                       // ================================================
                       // Proceed the reactive power for each phase
                       // ================================================
                       #Driver_Data.Q_L1_max := #V_DP_Meas_Min_Max.Q_L1_Max;
                       #Driver_Data.Q_L1_min := #V_DP_Meas_Min_Max.Q_L1_Min;
                       #Driver_Data.Q_L2_max := #V_DP_Meas_Min_Max.Q_L2_Max;
                       #Driver_Data.Q_L2_min := #V_DP_Meas_Min_Max.Q_L2_Min;
                       #Driver_Data.Q_L3_max := #V_DP_Meas_Min_Max.Q_L3_Max;
                       #Driver_Data.Q_L3_min := #V_DP_Meas_Min_Max.Q_L3_Min;
                       #Driver_Data.Q_Total_max := #V_DP_Meas_Min_Max.Q_Total_Max;
                       #Driver_Data.Q_Total_min := #V_DP_Meas_Min_Max.Q_Total_Min;

                       // ================================================
                       // Proceed the effective power for each phase
                       // ================================================
                       #Driver_Data.P_L1_max := #V_DP_Meas_Min_Max.P_L1_Max;
                       #Driver_Data.P_L1_min := #V_DP_Meas_Min_Max.P_L1_Min;
                       #Driver_Data.P_L2_max := #V_DP_Meas_Min_Max.P_L2_Max;
                       #Driver_Data.P_L2_min := #V_DP_Meas_Min_Max.P_L2_Min;
                       #Driver_Data.P_L3_max := #V_DP_Meas_Min_Max.P_L3_Max;
                       #Driver_Data.P_L3_min := #V_DP_Meas_Min_Max.P_L3_Min;
                       #Driver_Data.P_Total_max := #V_DP_Meas_Min_Max.P_Total_Max;
                       #Driver_Data.P_Total_min := #V_DP_Meas_Min_Max.P_Total_Min;

                       // Go back to the main state and wait for a new request
                       #Sm_State_Next := #SM_IDLE;
                   ELSE
                       ; // Reading still in progress
                   END_IF;
           END_CASE;

           // Set information for the visualization block
           #Driver_Data.Read_Value := #Automatic_Update;
           #Driver_Data.Driver_Error := BOOL_TO_INT(#Error_Code <> 0);
           #Driver_Data.Connection_Type := #Connection_Type;

           // Store the value for edge detection
           #Start_Acyclic_HMI_Old := #HMI_Bits_Internal.Start_Acyclic;
           #Reset_Energy_Old := #Reset_Energy_Counter;
           #Reset_Energy_HMI_Old := #HMI_Bits_Internal.Reset_Energy_Meter;
           #Reset_Min_Max_Old := #Reset_Min_Max;
           #Reset_Min_Max_HMI_Old := #HMI_Bits_Internal.Reset_min_max_Data;

       END_IF;
END_FUNCTION_BLOCK

FUNCTION_BLOCK "LProcPAC-Conversion"   // FB1743, SCL
TITLE = LProcPAC-Conversion
{ S7_Optimized_Access := 'TRUE' }
AUTHOR : CSTAAL
VERSION : 2.0
// stored: AutoNumber false, IsIECCheckEnabled false, IsRetainMemResEnabled false, MemoryReserve 100, SetENOAutomatically False, UDAEnableTagReadback false
   VAR_INPUT
      id_hdword { ExternalAccessible := 'False'; ExternalVisible := 'False'; ExternalWritable := 'False'} : DWord := DWORD#16#0000_0000;   // highdword of the 64Bit number
      id_ldword { ExternalAccessible := 'False'; ExternalVisible := 'False'; ExternalWritable := 'False'} : DWord := DWORD#16#0000_0000;   // lowdword of the 64Bit number
   END_VAR
   VAR_OUTPUT
      FINE { ExternalAccessible := 'False'; ExternalVisible := 'False'; ExternalWritable := 'False'} : DInt := 0;   // counter value fine
      RAW { ExternalAccessible := 'False'; ExternalVisible := 'False'; ExternalWritable := 'False'} : DInt := 0;   // counter value raw
      ERROR { ExternalAccessible := 'False'; ExternalVisible := 'False'; ExternalWritable := 'False'} : Word := WORD#16#0000;   // error word of the function block
   END_VAR
   VAR DB_SPECIFIC
      sCounterval { ExternalAccessible := 'False'; ExternalVisible := 'False'; ExternalWritable := 'False'} : Struct   // 64Bit structure
         hdword { ExternalAccessible := 'False'; ExternalVisible := 'False'; ExternalWritable := 'False'} : DWord := DWORD#16#0000_0000;   // highdword of the 64Bit number
         ldword { ExternalAccessible := 'False'; ExternalVisible := 'False'; ExternalWritable := 'False'} : DWord := DWORD#16#0000_0000;   // lowdword of the 64Bit number
      END_STRUCT;
   END_VAR
   VAR
      vwords AT sCounterval : Struct   // AT sCounterval : STRUCT
         HDHW : Word;   // highword of the highdword of the 64Bit number
         HDLW : Word;   // lowword of the highdword of the 64Bit number
         LDHW : Word;   // highword of the lowdword of the 64Bit number
         LDLW : Word;   // lowword of the lowdword of the 64Bit number
      END_STRUCT;
      sVZ { ExternalAccessible := 'False'; ExternalVisible := 'False'; ExternalWritable := 'False'} : Word := WORD#16#0000;   // algebraic sign of the 64Bit number
      sCH { ExternalAccessible := 'False'; ExternalVisible := 'False'; ExternalWritable := 'False'} : Word := WORD#16#0000;   // exponent of the 64Bit number
      sExp { ExternalAccessible := 'False'; ExternalVisible := 'False'; ExternalWritable := 'False'} : Int := 0;   // exponent of the 64Bit number
      sResDiv { ExternalAccessible := 'False'; ExternalVisible := 'False'; ExternalWritable := 'False'} : DWord := DWORD#16#0000_0000;   // result of division
      sDivision { ExternalAccessible := 'False'; ExternalVisible := 'False'; ExternalWritable := 'False'} : DWord := DWORD#16#0000_0000;   // dword for division of 1.000.000.000
      sFINE { ExternalAccessible := 'False'; ExternalVisible := 'False'; ExternalWritable := 'False'} : DInt := 0;   // static counter falue fine
      sRAW { ExternalAccessible := 'False'; ExternalVisible := 'False'; ExternalWritable := 'False'} : DInt := 0;   // static counter value raw
      sERROR { ExternalAccessible := 'False'; ExternalVisible := 'False'; ExternalWritable := 'False'} : Word := WORD#16#0000;   // static error word
      i { ExternalAccessible := 'False'; ExternalVisible := 'False'; ExternalWritable := 'False'} : Int := 0;   // loop counter
   END_VAR
   VAR CONSTANT
      cBIAS : Word := WORD#16#03FF;   // 03FFh --> 1023dez ... bias of the 64Bit number
      cVZmask : Word := WORD#16#8000;   // mask to seperate the algebraic sign
      cCHmask : Word := WORD#16#7FF0;   // mask to seperate the exponent field
      cMTmask : DWord := DWORD#16#000F_FFFF;   // mask to seperate the mantissa
      cMask : DWord := DWORD#16#0000_0001;   // general mask
      cNrGIGA : DInt := 1_000_000_000;   // 1.000.000.000(dez)
      cNrKILO : Int := 1000;   // 1.000(dez)
   END_VAR
BEGIN



   (***********************************************************************************************
   ********************************************  CODE  *******************************************
   ***********************************************************************************************)

   // initialization of internal variables
   // allocation of the two dwords of the energy counter value
   #sCounterval.hdword := #id_hdword;
   #sCounterval.ldword := #id_ldword;
   #sResDiv := dw#16#000000000;

   // seperate VZ (sign bit)
   #sVZ := #vwords.HDHW AND #cVZmask;

   // seperate CH (exponent field with offset(cBias))
   // seperate exponent of the 64Bit value
   #sCH := SHR(IN := (#vwords.HDHW AND #cCHmask), N := 4);
   #sExp := WORD_TO_INT(#sCH) - WORD_TO_INT(#cBIAS);

   // check the algebraic sign
   // negative counter values indicate an error
   IF #sVZ = #cVZmask
   THEN
       #sERROR := w#16#0001;
   ELSE
       // check the special case of the 0 value and the value < 1
       // the output values have the format dint --> 0,1 is not possible
       IF #sCH = w#16#0000 OR WORD_TO_INT(#sCH) < WORD_TO_INT(#cBIAS)
       THEN
           #sFINE := 0;
           #sRAW := 0;
       ELSE
           // **************************
           // ********** FINE **********
           // **************************

           // *** If the exponent is smaller than 29 the number is smaller than 1.000.000.000
           // *** You have to seperate the valid bits (sExp)of the mantissa
           // *** At the end you have to add the hidden 1 Bit
           IF #sExp < 29
           THEN
               IF #sExp < 20
               THEN
                   #sFINE := DWORD_TO_DINT(SHR(IN := (#sCounterval.hdword AND #cMTmask), N := 20 - #sExp) OR SHL(IN := #cMask, N := #sExp));

               ELSIF #sExp = 20
               THEN
                   #sFINE := DWORD_TO_DINT(#sCounterval.hdword AND #cMTmask OR SHL(IN := #cMask, N := 20));
               ELSE
                   #sFINE := DWORD_TO_DINT((SHL(IN := (#sCounterval.hdword AND #cMTmask), N := #sExp - 20) OR SHR(IN := #sCounterval.ldword, N := 32 - (#sExp - 20))) OR SHL(IN := #cMask, N := #sExp));
               END_IF;

               // *** If the exponent is 29 the number is between 536.870.912 and 1.073.741.823
               // *** You have to subtract 1.000.000.000 if it's bigger than 1.000.000.000
               // *** The result ist the fine counter value
           ELSIF #sExp = 29
           THEN
               IF DWORD_TO_DINT((SHL(IN := (#sCounterval.hdword AND #cMTmask), N := #sExp - 20) OR SHR(IN := #sCounterval.ldword, N := 32 - (#sExp - 20))) OR SHL(IN := #cMask, N := #sExp)) > #cNrGIGA
               THEN
                   #sFINE := DWORD_TO_DINT((SHL(IN := (#sCounterval.hdword AND #cMTmask), N := #sExp - 20) OR SHR(IN := #sCounterval.ldword, N := 32 - (#sExp - 20))) OR SHL(IN := #cMask, N := #sExp)) - #cNrGIGA;

               ELSIF DWORD_TO_DINT((SHL(IN := (#sCounterval.hdword AND #cMTmask), N := #sExp - 20) OR SHR(IN := #sCounterval.ldword, N := 32 - (#sExp - 20))) OR SHL(IN := #cMask, N := #sExp)) = #cNrGIGA
               THEN
                   #sFINE := 0;
               ELSE
                   #sFINE := DWORD_TO_DINT((SHL(IN := (#sCounterval.hdword AND #cMTmask), N := #sExp - 20) OR SHR(IN := #sCounterval.ldword, N := 32 - (#sExp - 20))) OR SHL(IN := #cMask, N := #sExp));
               END_IF;

               // *** If the exponent is bigger then 29 you have to divide the number by 1.000.000.000
               // *** the rest of the division is the fine counter value
           ELSE
               #sDivision := (SHL(IN := (#sCounterval.hdword AND #cMTmask), N := 9) OR SHR(IN := #sCounterval.ldword, N := 23)) OR SHL(IN := #cMask, N := 29);
               FOR #i := 0 TO #sExp - 29 DO
                   IF DWORD_TO_DINT(#sDivision) > #cNrGIGA OR DWORD_TO_DINT(#sDivision) = #cNrGIGA
                   THEN

                       #sDivision := DINT_TO_DWORD(DWORD_TO_DINT(#sDivision) - #cNrGIGA);
                       IF #i <> #sExp - 29
                       THEN
                           #sDivision := SHL(IN := #sDivision, N := 1) OR (SHR(IN := #sCounterval.ldword, N := 22 - #i) AND #cMask);
                       ELSE
                           ;
                       END_IF;

                       #sResDiv := SHL(IN := #sResDiv, N := 1) OR dw#16#00000001;
                   ELSE
                       IF #i <> #sExp - 29
                       THEN
                           #sDivision := SHL(IN := #sDivision, N := 1) OR (SHR(IN := #sCounterval.ldword, N := 22 - #i) AND #cMask);
                       ELSE
                           ;
                       END_IF;

                       #sResDiv := SHL(IN := #sResDiv, N := 1);
                   END_IF;

               END_FOR;

               #sFINE := DWORD_TO_DINT(#sDivision);

           END_IF;

           // **************************
           // ********** RAW ***********
           // **************************

           // Initialisation of sResDiv for new division
           #sResDiv := dw#16#00000000;

           // *** If the exponent is smaller than 9 the number is smaller than 1.000
           // *** The raw counter value is 0
           IF #sExp < 9
           THEN
               #sRAW := 0;

               // *** If the exponent is 9 the number is between 512 and 1.023
               // *** You have to subtract 1.000
               // *** The result ist the raw counter value
           ELSIF #sExp = 9
           THEN
               IF DWORD_TO_DINT(SHR(IN := (#sCounterval.hdword AND #cMTmask), N := 20 - #sExp) OR SHL(IN := #cMask, N := #sExp)) > #cNrKILO
               THEN
                   #sRAW := 1;
               ELSE
                   #sRAW := 0;
               END_IF;

               // *** If the exponent is bigger then 29 you have to divide the number by 1.000.000.000
               // *** the result of the division is the raw countervalue
           ELSE
               #sDivision := SHR(IN := (#sCounterval.hdword AND #cMTmask), N := 11) OR SHL(IN := #cMask, N := 9);
               FOR #i := 0 TO #sExp - 9 DO
                   IF DWORD_TO_DINT(#sDivision) > #cNrKILO OR DWORD_TO_DINT(#sDivision) = #cNrKILO
                   THEN

                       #sDivision := DINT_TO_DWORD(DWORD_TO_DINT(#sDivision) - #cNrKILO);
                       IF #i <> #sExp - 9
                       THEN
                           #sDivision := SHL(IN := #sDivision, N := 1);
                           IF #i <= 10
                           THEN
                               #sDivision := #sDivision OR (SHR(IN := #sCounterval.hdword, N := 11 - (#i + 1)) AND #cMask);
                           ELSE
                               #sDivision := #sDivision OR (SHR(IN := #sCounterval.ldword, N := 32 - ((#i + 1) - 11)) AND #cMask);
                           END_IF;

                       ELSE
                           ;
                       END_IF;

                       #sResDiv := SHL(IN := #sResDiv, N := 1) OR dw#16#00000001;
                   ELSE
                       IF #i <> #sExp - 9
                       THEN
                           #sDivision := SHL(IN := #sDivision, N := 1);
                           IF #i <= 10
                           THEN
                               #sDivision := #sDivision OR (SHR(IN := #sCounterval.hdword, N := 11 - (#i + 1)) AND #cMask);
                           ELSE
                               #sDivision := #sDivision OR (SHR(IN := #sCounterval.ldword, N := 32 - ((#i + 1) - 11)) AND #cMask);
                           END_IF;

                       ELSE
                           ;
                       END_IF;

                       #sResDiv := SHL(IN := #sResDiv, N := 1);
                   END_IF;

               END_FOR;

               #sRAW := DWORD_TO_DINT(#sResDiv);

           END_IF;

       END_IF;
       #sERROR := w#16#0000;
   END_IF;

   #FINE := #sFINE;
   #RAW := #sRAW;
   #ERROR := #sERROR;
END_FUNCTION_BLOCK

FUNCTION_BLOCK "LProcPAC-Visu"   // FB1742, SCL
TITLE = LProcPAC-Visu
{ S7_Optimized_Access := 'FALSE' }
AUTHOR : CSTAAL
VERSION : 2.0
// 20131213
// ======================================================================================================================
// ==========Short Description===========================================================================================
// ======================================================================================================================
// 
//   This function block is a interface between driver function block and WinCC. 
//   
// ======================================================================================================================
// ==========Dependencies(Abhängigkeit)==================================================================================
// ======================================================================================================================
// 
//   none
// 
// ======================================================================================================================
// ==========Change Log==================================================================================================
// ======================================================================================================================
// 
//       DATE    |   Version     |   NAME        |   CHANGE
//   ------------|---------------|---------------|--------------------------
//               |   v1.0        |   DirkTie     |   - First implementation 
//   ------------|---------------|---------------|--------------------------
//               |   v2.0        |   BaueChr     |   - bug fixes 
//   ------------|---------------|---------------|--------------------------
// 
// ======================================================================================================================
// ==========Know Issues=================================================================================================
// ======================================================================================================================
// 
//     - v2.0:
//             wrong connections of the energy counters to the outputs                 ... fixed 2014/08/22
//             extent the automatic change of the current unit over all phases            ... fixed 2014/08/22
//             extent driver_data structure (Connection_Type & Driver_error)            ... fixed 2014/08/22
//             change constant MAX_VALUE to 750 to define the correct scale end value    ... fixed 2014/08/25
//             new definition of the scale start value of reactive power if Qmin > 0    ... fixed 2014/08/25
// 
// ======================================================================================================================
// ==========Constant Definitions========================================================================================
// ======================================================================================================================
// stored: AutoNumber false, IsIECCheckEnabled false, SetENOAutomatically False, UDAEnableTagReadback false
   VAR_INPUT
      Add_Value_Count { ExternalAccessible := 'False'; ExternalVisible := 'False'; ExternalWritable := 'False'} : Int := 0;   // count of the user measurements
      AddValue_01 { ExternalAccessible := 'False'; ExternalVisible := 'False'; ExternalWritable := 'False'} : Real := 0.0;   // user measurements 01
      AddValue_02 { ExternalAccessible := 'False'; ExternalVisible := 'False'; ExternalWritable := 'False'} : Real := 0.0;   // user measurements 02
      AddValue_03 { ExternalAccessible := 'False'; ExternalVisible := 'False'; ExternalWritable := 'False'} : Real := 0.0;   // user measurements 03
      AddValue_04 { ExternalAccessible := 'False'; ExternalVisible := 'False'; ExternalWritable := 'False'} : Real := 0.0;   // user measurements 04
      AddValue_05 { ExternalAccessible := 'False'; ExternalVisible := 'False'; ExternalWritable := 'False'} : Real := 0.0;   // user measurements 05
      AddValue_06 { ExternalAccessible := 'False'; ExternalVisible := 'False'; ExternalWritable := 'False'} : Real := 0.0;   // user measurements 06
      AddValue_07 { ExternalAccessible := 'False'; ExternalVisible := 'False'; ExternalWritable := 'False'} : Real := 0.0;   // user measurements 07
      AddValue_08 { ExternalAccessible := 'False'; ExternalVisible := 'False'; ExternalWritable := 'False'} : Real := 0.0;   // user measurements 08
      AddValue_09 { ExternalAccessible := 'False'; ExternalVisible := 'False'; ExternalWritable := 'False'} : Real := 0.0;   // user measurements 09
      AddValue_10 { ExternalAccessible := 'False'; ExternalVisible := 'False'; ExternalWritable := 'False'} : Real := 0.0;   // user measurements 10
      AddValue_11 { ExternalAccessible := 'False'; ExternalVisible := 'False'; ExternalWritable := 'False'} : Real := 0.0;   // user measurements 11
      AddValue_12 { ExternalAccessible := 'False'; ExternalVisible := 'False'; ExternalWritable := 'False'} : Real := 0.0;   // user measurements 12
      Start_Acyclic { ExternalAccessible := 'False'; ExternalVisible := 'False'; ExternalWritable := 'False'} : Bool := FALSE;
      Start_Auto { ExternalAccessible := 'False'; ExternalVisible := 'False'; ExternalWritable := 'False'} : Bool := FALSE;
      Reset_min_max_Data { ExternalAccessible := 'False'; ExternalVisible := 'False'; ExternalWritable := 'False'} : Bool := FALSE;
      Reset_Energy_Meter { ExternalAccessible := 'False'; ExternalVisible := 'False'; ExternalWritable := 'False'} : Bool := FALSE;   // ================================================================================================================================inoutput variablen================================================================================================================================================================================================================
   END_VAR
   VAR_OUTPUT
      U_L1_L2 { ExternalAccessible := 'False'; ExternalVisible := 'False'; ExternalWritable := 'False'} : Real := 0.0;   // voltage L1-L2
      U_L2_L3 { ExternalAccessible := 'False'; ExternalVisible := 'False'; ExternalWritable := 'False'} : Real := 0.0;   // voltage L2-L3
      U_L3_L1 { ExternalAccessible := 'False'; ExternalVisible := 'False'; ExternalWritable := 'False'} : Real := 0.0;   // voltage L3-L1
      U_L1 { ExternalAccessible := 'False'; ExternalVisible := 'False'; ExternalWritable := 'False'} : Real := 0.0;   // voltage L1-N
      U_L2 { ExternalAccessible := 'False'; ExternalVisible := 'False'; ExternalWritable := 'False'} : Real := 0.0;   // voltage L2-N
      U_L3 { ExternalAccessible := 'False'; ExternalVisible := 'False'; ExternalWritable := 'False'} : Real := 0.0;   // voltage L3-N
      U_L1_L2_min { ExternalAccessible := 'False'; ExternalVisible := 'False'; ExternalWritable := 'False'} : Real := 0.0;   // minimum voltage U1
      U_L2_L3_min { ExternalAccessible := 'False'; ExternalVisible := 'False'; ExternalWritable := 'False'} : Real := 0.0;   // minimum voltage U2
      U_L3_L1_min { ExternalAccessible := 'False'; ExternalVisible := 'False'; ExternalWritable := 'False'} : Real := 0.0;
      U_L1_min { ExternalAccessible := 'False'; ExternalVisible := 'False'; ExternalWritable := 'False'} : Real := 0.0;   // minimum voltage U1
      U_L2_min { ExternalAccessible := 'False'; ExternalVisible := 'False'; ExternalWritable := 'False'} : Real := 0.0;   // minimum voltage U2
      U_L3_min { ExternalAccessible := 'False'; ExternalVisible := 'False'; ExternalWritable := 'False'} : Real := 0.0;   // minimum voltage U3
      U_L1_L2_max { ExternalAccessible := 'False'; ExternalVisible := 'False'; ExternalWritable := 'False'} : Real := 0.0;   // maximum voltage U1
      U_L2_L3_max { ExternalAccessible := 'False'; ExternalVisible := 'False'; ExternalWritable := 'False'} : Real := 0.0;   // maximum voltage U2
      U_L3_L1_max { ExternalAccessible := 'False'; ExternalVisible := 'False'; ExternalWritable := 'False'} : Real := 0.0;   // maximum voltage U3
      U_L1_max { ExternalAccessible := 'False'; ExternalVisible := 'False'; ExternalWritable := 'False'} : Real := 0.0;   // maximum voltage U1
      U_L2_max { ExternalAccessible := 'False'; ExternalVisible := 'False'; ExternalWritable := 'False'} : Real := 0.0;   // maximum voltage U2
      U_L3_max { ExternalAccessible := 'False'; ExternalVisible := 'False'; ExternalWritable := 'False'} : Real := 0.0;   // maximum voltage U3
      U_PH_PH_Average { ExternalAccessible := 'False'; ExternalVisible := 'False'; ExternalWritable := 'False'} : Real := 0.0;   // averagevoltage PH-PH
      U_PH_N_Average { ExternalAccessible := 'False'; ExternalVisible := 'False'; ExternalWritable := 'False'} : Real := 0.0;   // averagevoltage PH-N
      U_PH_PH_Average_min { ExternalAccessible := 'False'; ExternalVisible := 'False'; ExternalWritable := 'False'} : Real := 0.0;   // minimum averagevoltage PH-PH
      U_PH_N_Average_min { ExternalAccessible := 'False'; ExternalVisible := 'False'; ExternalWritable := 'False'} : Real := 0.0;   // minimum averagevoltage PH-N
      U_PH_PH_Average_max { ExternalAccessible := 'False'; ExternalVisible := 'False'; ExternalWritable := 'False'} : Real := 0.0;   // maximum averagevoltage PH-PH
      U_PH_N_Average_max { ExternalAccessible := 'False'; ExternalVisible := 'False'; ExternalWritable := 'False'} : Real := 0.0;   // maximum averagevoltage PH-N
      I_L1 { ExternalAccessible := 'False'; ExternalVisible := 'False'; ExternalWritable := 'False'} : Real := 0.0;   // current I1
      I_L2 { ExternalAccessible := 'False'; ExternalVisible := 'False'; ExternalWritable := 'False'} : Real := 0.0;   // current I2
      I_L3 { ExternalAccessible := 'False'; ExternalVisible := 'False'; ExternalWritable := 'False'} : Real := 0.0;   // current I3
      I_L1_min { ExternalAccessible := 'False'; ExternalVisible := 'False'; ExternalWritable := 'False'} : Real := 0.0;   // minimum current I1
      I_L2_min { ExternalAccessible := 'False'; ExternalVisible := 'False'; ExternalWritable := 'False'} : Real := 0.0;   // minimum current I2
      I_L3_min { ExternalAccessible := 'False'; ExternalVisible := 'False'; ExternalWritable := 'False'} : Real := 0.0;   // minimum current I3
      I_L1_max { ExternalAccessible := 'False'; ExternalVisible := 'False'; ExternalWritable := 'False'} : Real := 0.0;   // maximum current I1
      I_L2_max { ExternalAccessible := 'False'; ExternalVisible := 'False'; ExternalWritable := 'False'} : Real := 0.0;   // maximum current I2
      I_L3_max { ExternalAccessible := 'False'; ExternalVisible := 'False'; ExternalWritable := 'False'} : Real := 0.0;   // maximum current I3
      I_Average { ExternalAccessible := 'False'; ExternalVisible := 'False'; ExternalWritable := 'False'} : Real := 0.0;   // average currentI
      I_Average_min { ExternalAccessible := 'False'; ExternalVisible := 'False'; ExternalWritable := 'False'} : Real := 0.0;   // minimum average currentI
      I_Average_max { ExternalAccessible := 'False'; ExternalVisible := 'False'; ExternalWritable := 'False'} : Real := 0.0;   // maximum average currentI
      f { ExternalAccessible := 'False'; ExternalVisible := 'False'; ExternalWritable := 'False'} : Real := 0.0;   // frequency
      f_min { ExternalAccessible := 'False'; ExternalVisible := 'False'; ExternalWritable := 'False'} : Real := 0.0;   // minimum frequency
      f_max { ExternalAccessible := 'False'; ExternalVisible := 'False'; ExternalWritable := 'False'} : Real := 0.0;   // maximum frequency
      S_Total { ExternalAccessible := 'False'; ExternalVisible := 'False'; ExternalWritable := 'False'} : Real := 0.0;   // total apparent power
      S_Total_min { ExternalAccessible := 'False'; ExternalVisible := 'False'; ExternalWritable := 'False'} : Real := 0.0;   // minimum total apparent power
      S_Total_max { ExternalAccessible := 'False'; ExternalVisible := 'False'; ExternalWritable := 'False'} : Real := 0.0;   // maximum total apparent power
      P_Total { ExternalAccessible := 'False'; ExternalVisible := 'False'; ExternalWritable := 'False'} : Real := 0.0;   // total active power
      P_Total_min { ExternalAccessible := 'False'; ExternalVisible := 'False'; ExternalWritable := 'False'} : Real := 0.0;   // minimum total active power
      P_Total_max { ExternalAccessible := 'False'; ExternalVisible := 'False'; ExternalWritable := 'False'} : Real := 0.0;   // maximum total active power
      Q_Total { ExternalAccessible := 'False'; ExternalVisible := 'False'; ExternalWritable := 'False'} : Real := 0.0;   // total reactive power
      Q_Total_min { ExternalAccessible := 'False'; ExternalVisible := 'False'; ExternalWritable := 'False'} : Real := 0.0;   // minimum total reactive power
      Q_Total_max { ExternalAccessible := 'False'; ExternalVisible := 'False'; ExternalWritable := 'False'} : Real := 0.0;   // maximum total reactive power
      Cos_Total { ExternalAccessible := 'False'; ExternalVisible := 'False'; ExternalWritable := 'False'} : Real := 0.0;   // total efficiency factor
      Cos_Total_min { ExternalAccessible := 'False'; ExternalVisible := 'False'; ExternalWritable := 'False'} : Real := 0.0;   // minimum total efficiency factor
      Cos_Total_max { ExternalAccessible := 'False'; ExternalVisible := 'False'; ExternalWritable := 'False'} : Real := 0.0;   // maximum total efficiency factor
      Cos_L1 { ExternalAccessible := 'False'; ExternalVisible := 'False'; ExternalWritable := 'False'} : Real := 0.0;   // efficiency factor L1
      Cos_L1_min { ExternalAccessible := 'False'; ExternalVisible := 'False'; ExternalWritable := 'False'} : Real := 0.0;   // minimum efficiency factor L1
      Cos_L1_max { ExternalAccessible := 'False'; ExternalVisible := 'False'; ExternalWritable := 'False'} : Real := 0.0;   // maximum efficiency factor L1
      Cos_L2 { ExternalAccessible := 'False'; ExternalVisible := 'False'; ExternalWritable := 'False'} : Real := 0.0;   // efficiency factor L2
      Cos_L2_min { ExternalAccessible := 'False'; ExternalVisible := 'False'; ExternalWritable := 'False'} : Real := 0.0;   // minimum efficiency factor L2
      Cos_L2_max { ExternalAccessible := 'False'; ExternalVisible := 'False'; ExternalWritable := 'False'} : Real := 0.0;   // maximum efficiency factor L2
      Cos_L3 { ExternalAccessible := 'False'; ExternalVisible := 'False'; ExternalWritable := 'False'} : Real := 0.0;   // efficiency factor L3
      Cos_L3_min { ExternalAccessible := 'False'; ExternalVisible := 'False'; ExternalWritable := 'False'} : Real := 0.0;   // minimum efficiency factor L3
      Cos_Total_1 { ExternalAccessible := 'False'; ExternalVisible := 'False'; ExternalWritable := 'False'} : Real;
      Cos_Total_min_1 { ExternalAccessible := 'False'; ExternalVisible := 'False'; ExternalWritable := 'False'} : Real;
      Cos_Total_max_1 { ExternalAccessible := 'False'; ExternalVisible := 'False'; ExternalWritable := 'False'} : Real;
      Cos_L2_1 { ExternalAccessible := 'False'; ExternalVisible := 'False'; ExternalWritable := 'False'} : Real;
      Cos_L1_min_1 { ExternalAccessible := 'False'; ExternalVisible := 'False'; ExternalWritable := 'False'} : Real;
      Cos_L1_max_1 { ExternalAccessible := 'False'; ExternalVisible := 'False'; ExternalWritable := 'False'} : Real;
      Cos_L3_1 { ExternalAccessible := 'False'; ExternalVisible := 'False'; ExternalWritable := 'False'} : Real;
      Cos_L2_min_1 { ExternalAccessible := 'False'; ExternalVisible := 'False'; ExternalWritable := 'False'} : Real;
      Cos_L2_max_1 { ExternalAccessible := 'False'; ExternalVisible := 'False'; ExternalWritable := 'False'} : Real;
      Cos_L4 { ExternalAccessible := 'False'; ExternalVisible := 'False'; ExternalWritable := 'False'} : Real;
      Cos_L3_min_1 { ExternalAccessible := 'False'; ExternalVisible := 'False'; ExternalWritable := 'False'} : Real;
      Cos_Total_2 { ExternalAccessible := 'False'; ExternalVisible := 'False'; ExternalWritable := 'False'} : Real;
      Cos_Total_min_2 { ExternalAccessible := 'False'; ExternalVisible := 'False'; ExternalWritable := 'False'} : Real;
      Cos_Total_max_2 { ExternalAccessible := 'False'; ExternalVisible := 'False'; ExternalWritable := 'False'} : Real;
      Cos_L3_2 { ExternalAccessible := 'False'; ExternalVisible := 'False'; ExternalWritable := 'False'} : Real;
      Cos_L1_min_2 { ExternalAccessible := 'False'; ExternalVisible := 'False'; ExternalWritable := 'False'} : Real;
      Cos_L1_max_2 { ExternalAccessible := 'False'; ExternalVisible := 'False'; ExternalWritable := 'False'} : Real;
      Cos_L4_1 { ExternalAccessible := 'False'; ExternalVisible := 'False'; ExternalWritable := 'False'} : Real;
      Cos_L2_min_2 { ExternalAccessible := 'False'; ExternalVisible := 'False'; ExternalWritable := 'False'} : Real;
      Cos_L2_max_2 { ExternalAccessible := 'False'; ExternalVisible := 'False'; ExternalWritable := 'False'} : Real;
      Cos_L5 { ExternalAccessible := 'False'; ExternalVisible := 'False'; ExternalWritable := 'False'} : Real;
      Cos_L3_min_2 { ExternalAccessible := 'False'; ExternalVisible := 'False'; ExternalWritable := 'False'} : Real;
      Cos_Total_3 { ExternalAccessible := 'False'; ExternalVisible := 'False'; ExternalWritable := 'False'} : Real;
      Cos_Total_min_3 { ExternalAccessible := 'False'; ExternalVisible := 'False'; ExternalWritable := 'False'} : Real;
      Cos_Total_max_3 { ExternalAccessible := 'False'; ExternalVisible := 'False'; ExternalWritable := 'False'} : Real;
      Cos_L4_2 { ExternalAccessible := 'False'; ExternalVisible := 'False'; ExternalWritable := 'False'} : Real;
      Cos_L1_min_3 { ExternalAccessible := 'False'; ExternalVisible := 'False'; ExternalWritable := 'False'} : Real;
      Cos_L1_max_3 { ExternalAccessible := 'False'; ExternalVisible := 'False'; ExternalWritable := 'False'} : Real;
      Cos_L5_1 { ExternalAccessible := 'False'; ExternalVisible := 'False'; ExternalWritable := 'False'} : Real;
      Cos_L2_min_3 { ExternalAccessible := 'False'; ExternalVisible := 'False'; ExternalWritable := 'False'} : Real;
      Cos_L2_max_3 { ExternalAccessible := 'False'; ExternalVisible := 'False'; ExternalWritable := 'False'} : Real;
      Cos_L6 { ExternalAccessible := 'False'; ExternalVisible := 'False'; ExternalWritable := 'False'} : Real;
      Cos_L3_min_3 { ExternalAccessible := 'False'; ExternalVisible := 'False'; ExternalWritable := 'False'} : Real;
      Cos_Total_4 { ExternalAccessible := 'False'; ExternalVisible := 'False'; ExternalWritable := 'False'} : Real;
      Cos_Total_min_4 { ExternalAccessible := 'False'; ExternalVisible := 'False'; ExternalWritable := 'False'} : Real;
      Cos_Total_max_4 { ExternalAccessible := 'False'; ExternalVisible := 'False'; ExternalWritable := 'False'} : Real;
      Cos_L5_2 { ExternalAccessible := 'False'; ExternalVisible := 'False'; ExternalWritable := 'False'} : Real;
      Cos_L1_min_4 { ExternalAccessible := 'False'; ExternalVisible := 'False'; ExternalWritable := 'False'} : Real;
      Cos_L1_max_4 { ExternalAccessible := 'False'; ExternalVisible := 'False'; ExternalWritable := 'False'} : Real;
      Cos_L6_1 { ExternalAccessible := 'False'; ExternalVisible := 'False'; ExternalWritable := 'False'} : Real;
      Cos_L2_min_4 { ExternalAccessible := 'False'; ExternalVisible := 'False'; ExternalWritable := 'False'} : Real;
      Cos_L2_max_4 { ExternalAccessible := 'False'; ExternalVisible := 'False'; ExternalWritable := 'False'} : Real;
      Cos_L7 { ExternalAccessible := 'False'; ExternalVisible := 'False'; ExternalWritable := 'False'} : Real;
      Cos_L3_min_4 { ExternalAccessible := 'False'; ExternalVisible := 'False'; ExternalWritable := 'False'} : Real;
      Cos_Total_5 { ExternalAccessible := 'False'; ExternalVisible := 'False'; ExternalWritable := 'False'} : Real;
      Cos_Total_min_5 { ExternalAccessible := 'False'; ExternalVisible := 'False'; ExternalWritable := 'False'} : Real;
      Cos_Total_max_5 { ExternalAccessible := 'False'; ExternalVisible := 'False'; ExternalWritable := 'False'} : Real;
      Cos_L6_2 { ExternalAccessible := 'False'; ExternalVisible := 'False'; ExternalWritable := 'False'} : Real;
      Cos_L1_min_5 { ExternalAccessible := 'False'; ExternalVisible := 'False'; ExternalWritable := 'False'} : Real;
      Cos_L1_max_5 { ExternalAccessible := 'False'; ExternalVisible := 'False'; ExternalWritable := 'False'} : Real;
      Cos_L7_1 { ExternalAccessible := 'False'; ExternalVisible := 'False'; ExternalWritable := 'False'} : Real;
      Cos_L2_min_5 { ExternalAccessible := 'False'; ExternalVisible := 'False'; ExternalWritable := 'False'} : Real;
      Cos_L2_max_5 { ExternalAccessible := 'False'; ExternalVisible := 'False'; ExternalWritable := 'False'} : Real;
      Cos_L8 { ExternalAccessible := 'False'; ExternalVisible := 'False'; ExternalWritable := 'False'} : Real;
      Cos_L3_min_5 { ExternalAccessible := 'False'; ExternalVisible := 'False'; ExternalWritable := 'False'} : Real;
      Cos_Total_6 { ExternalAccessible := 'False'; ExternalVisible := 'False'; ExternalWritable := 'False'} : Real;
      Cos_Total_min_6 { ExternalAccessible := 'False'; ExternalVisible := 'False'; ExternalWritable := 'False'} : Real;
      Cos_Total_max_6 { ExternalAccessible := 'False'; ExternalVisible := 'False'; ExternalWritable := 'False'} : Real;
      Cos_L7_2 { ExternalAccessible := 'False'; ExternalVisible := 'False'; ExternalWritable := 'False'} : Real;
      Cos_L1_min_6 { ExternalAccessible := 'False'; ExternalVisible := 'False'; ExternalWritable := 'False'} : Real;
      Cos_L1_max_6 { ExternalAccessible := 'False'; ExternalVisible := 'False'; ExternalWritable := 'False'} : Real;
      Cos_L8_1 { ExternalAccessible := 'False'; ExternalVisible := 'False'; ExternalWritable := 'False'} : Real;
      Cos_L2_min_6 { ExternalAccessible := 'False'; ExternalVisible := 'False'; ExternalWritable := 'False'} : Real;
      Cos_L2_max_6 { ExternalAccessible := 'False'; ExternalVisible := 'False'; ExternalWritable := 'False'} : Real;
      Cos_L9 { ExternalAccessible := 'False'; ExternalVisible := 'False'; ExternalWritable := 'False'} : Real;
      Cos_L3_min_6 { ExternalAccessible := 'False'; ExternalVisible := 'False'; ExternalWritable := 'False'} : Real;
      Cos_Total_7 { ExternalAccessible := 'False'; ExternalVisible := 'False'; ExternalWritable := 'False'} : Real;
      Cos_Total_min_7 { ExternalAccessible := 'False'; ExternalVisible := 'False'; ExternalWritable := 'False'} : Real;
      Cos_Total_max_7 { ExternalAccessible := 'False'; ExternalVisible := 'False'; ExternalWritable := 'False'} : Real;
      Cos_L8_2 { ExternalAccessible := 'False'; ExternalVisible := 'False'; ExternalWritable := 'False'} : Real;
      Cos_L1_min_7 { ExternalAccessible := 'False'; ExternalVisible := 'False'; ExternalWritable := 'False'} : Real;
      Cos_L1_max_7 { ExternalAccessible := 'False'; ExternalVisible := 'False'; ExternalWritable := 'False'} : Real;
      Cos_L9_1 { ExternalAccessible := 'False'; ExternalVisible := 'False'; ExternalWritable := 'False'} : Real;
      Cos_L2_min_7 { ExternalAccessible := 'False'; ExternalVisible := 'False'; ExternalWritable := 'False'} : Real;
      Cos_L2_max_7 { ExternalAccessible := 'False'; ExternalVisible := 'False'; ExternalWritable := 'False'} : Real;
      Cos_L10 { ExternalAccessible := 'False'; ExternalVisible := 'False'; ExternalWritable := 'False'} : Real;
      Cos_L3_min_7 { ExternalAccessible := 'False'; ExternalVisible := 'False'; ExternalWritable := 'False'} : Real;
      Cos_Total_8 { ExternalAccessible := 'False'; ExternalVisible := 'False'; ExternalWritable := 'False'} : Real;
      Cos_Total_min_8 { ExternalAccessible := 'False'; ExternalVisible := 'False'; ExternalWritable := 'False'} : Real;
      Cos_Total_max_8 { ExternalAccessible := 'False'; ExternalVisible := 'False'; ExternalWritable := 'False'} : Real;
      Cos_L9_2 { ExternalAccessible := 'False'; ExternalVisible := 'False'; ExternalWritable := 'False'} : Real;
      Cos_L1_min_8 { ExternalAccessible := 'False'; ExternalVisible := 'False'; ExternalWritable := 'False'} : Real;
      Cos_L1_max_8 { ExternalAccessible := 'False'; ExternalVisible := 'False'; ExternalWritable := 'False'} : Real;
      Cos_L10_1 { ExternalAccessible := 'False'; ExternalVisible := 'False'; ExternalWritable := 'False'} : Real;
      Cos_L2_min_8 { ExternalAccessible := 'False'; ExternalVisible := 'False'; ExternalWritable := 'False'} : Real;
      Cos_L2_max_8 { ExternalAccessible := 'False'; ExternalVisible := 'False'; ExternalWritable := 'False'} : Real;
      Cos_L11 { ExternalAccessible := 'False'; ExternalVisible := 'False'; ExternalWritable := 'False'} : Real;
      Cos_L3_min_8 { ExternalAccessible := 'False'; ExternalVisible := 'False'; ExternalWritable := 'False'} : Real;
      Cos_Total_9 { ExternalAccessible := 'False'; ExternalVisible := 'False'; ExternalWritable := 'False'} : Real;
      Cos_Total_min_9 { ExternalAccessible := 'False'; ExternalVisible := 'False'; ExternalWritable := 'False'} : Real;
      Cos_Total_max_9 { ExternalAccessible := 'False'; ExternalVisible := 'False'; ExternalWritable := 'False'} : Real;
      Cos_L10_2 { ExternalAccessible := 'False'; ExternalVisible := 'False'; ExternalWritable := 'False'} : Real;
      Cos_L1_min_9 { ExternalAccessible := 'False'; ExternalVisible := 'False'; ExternalWritable := 'False'} : Real;
      Cos_L1_max_9 { ExternalAccessible := 'False'; ExternalVisible := 'False'; ExternalWritable := 'False'} : Real;
      Cos_L11_1 { ExternalAccessible := 'False'; ExternalVisible := 'False'; ExternalWritable := 'False'} : Real;
      Cos_L3_max { ExternalAccessible := 'False'; ExternalVisible := 'False'; ExternalWritable := 'False'} : Real := 0.0;   // maximum efficiency factor L3
      S_L1 { ExternalAccessible := 'False'; ExternalVisible := 'False'; ExternalWritable := 'False'} : Real := 0.0;   // apparent power S1
      S_L2 { ExternalAccessible := 'False'; ExternalVisible := 'False'; ExternalWritable := 'False'} : Real := 0.0;   // apparent power S2
      S_L3 { ExternalAccessible := 'False'; ExternalVisible := 'False'; ExternalWritable := 'False'} : Real := 0.0;   // apparent power S3
      S_L1_min { ExternalAccessible := 'False'; ExternalVisible := 'False'; ExternalWritable := 'False'} : Real := 0.0;   // minimum apparent power S1
      S_L2_min { ExternalAccessible := 'False'; ExternalVisible := 'False'; ExternalWritable := 'False'} : Real := 0.0;   // minimum apparent power S2
      S_L3_min { ExternalAccessible := 'False'; ExternalVisible := 'False'; ExternalWritable := 'False'} : Real := 0.0;   // minimum apparent power S3
      S_L1_max { ExternalAccessible := 'False'; ExternalVisible := 'False'; ExternalWritable := 'False'} : Real := 0.0;   // maximum apparent power S1
      S_L2_max { ExternalAccessible := 'False'; ExternalVisible := 'False'; ExternalWritable := 'False'} : Real := 0.0;   // maximum apparent power S2
      S_L3_max { ExternalAccessible := 'False'; ExternalVisible := 'False'; ExternalWritable := 'False'} : Real := 0.0;   // maximum apparent power S3
      P_L1 { ExternalAccessible := 'False'; ExternalVisible := 'False'; ExternalWritable := 'False'} : Real := 0.0;   // reactive active power P1
      P_L2 { ExternalAccessible := 'False'; ExternalVisible := 'False'; ExternalWritable := 'False'} : Real := 0.0;   // reactive active power P2
      P_L3 { ExternalAccessible := 'False'; ExternalVisible := 'False'; ExternalWritable := 'False'} : Real := 0.0;   // reactive active power P3
      P_L1_min { ExternalAccessible := 'False'; ExternalVisible := 'False'; ExternalWritable := 'False'} : Real := 0.0;   // minimum active power P1
      P_L2_min { ExternalAccessible := 'False'; ExternalVisible := 'False'; ExternalWritable := 'False'} : Real := 0.0;   // minimum active power P2
      P_L3_min { ExternalAccessible := 'False'; ExternalVisible := 'False'; ExternalWritable := 'False'} : Real := 0.0;   // minimum active power P3
      P_L1_max { ExternalAccessible := 'False'; ExternalVisible := 'False'; ExternalWritable := 'False'} : Real := 0.0;   // maximum active power P1
      P_L2_max { ExternalAccessible := 'False'; ExternalVisible := 'False'; ExternalWritable := 'False'} : Real := 0.0;   // maximum active power P2
      P_L3_max { ExternalAccessible := 'False'; ExternalVisible := 'False'; ExternalWritable := 'False'} : Real := 0.0;   // maximum active power P3
      Q_L1 { ExternalAccessible := 'False'; ExternalVisible := 'False'; ExternalWritable := 'False'} : Real := 0.0;   // reactive_power Q1
      Q_L2 { ExternalAccessible := 'False'; ExternalVisible := 'False'; ExternalWritable := 'False'} : Real := 0.0;   // reactive_power Q2
      Q_L3 { ExternalAccessible := 'False'; ExternalVisible := 'False'; ExternalWritable := 'False'} : Real := 0.0;   // reactive_power Q3
      Q_L1_min { ExternalAccessible := 'False'; ExternalVisible := 'False'; ExternalWritable := 'False'} : Real := 0.0;   // minimum reactive_power Q1
      Q_L2_min { ExternalAccessible := 'False'; ExternalVisible := 'False'; ExternalWritable := 'False'} : Real := 0.0;   // minimum reactive_power Q2
      Q_L3_min { ExternalAccessible := 'False'; ExternalVisible := 'False'; ExternalWritable := 'False'} : Real := 0.0;   // minimum reactive_power Q3
      Q_L1_max { ExternalAccessible := 'False'; ExternalVisible := 'False'; ExternalWritable := 'False'} : Real := 0.0;   // maximum reactive_power Q1
      Q_L2_max { ExternalAccessible := 'False'; ExternalVisible := 'False'; ExternalWritable := 'False'} : Real := 0.0;   // maximum reactive_power Q2
      Q_L3_max { ExternalAccessible := 'False'; ExternalVisible := 'False'; ExternalWritable := 'False'} : Real := 0.0;   // maximum reactive_power Q3
      E_Active_Rate1_Import { ExternalAccessible := 'False'; ExternalVisible := 'False'; ExternalWritable := 'False'} : Real := 0.0;   // energy meter active power use rate1
      E_Active_Rate2_Import { ExternalAccessible := 'False'; ExternalVisible := 'False'; ExternalWritable := 'False'} : Real := 0.0;   // energy meter active power use rate2
      E_Active_Rate1_Export { ExternalAccessible := 'False'; ExternalVisible := 'False'; ExternalWritable := 'False'} : Real := 0.0;   // energy meter active power export rate1
      E_Active_Rate2_Export { ExternalAccessible := 'False'; ExternalVisible := 'False'; ExternalWritable := 'False'} : Real := 0.0;   // energy meter active power export rate2
      E_Reactive_Rate1_Import { ExternalAccessible := 'False'; ExternalVisible := 'False'; ExternalWritable := 'False'} : Real := 0.0;   // energy meter reactive power use rate1
      E_Reactive_Rate2_Import { ExternalAccessible := 'False'; ExternalVisible := 'False'; ExternalWritable := 'False'} : Real := 0.0;   // energy meter reactive power use rate2
      E_Reactive_Rate1_Export { ExternalAccessible := 'False'; ExternalVisible := 'False'; ExternalWritable := 'False'} : Real := 0.0;   // energy meter reactive power export rate1
      E_Reactive_Rate2_Export { ExternalAccessible := 'False'; ExternalVisible := 'False'; ExternalWritable := 'False'} : Real := 0.0;   // energy meter reactive power export rate2
      E_Apparent_Rate1_Import { ExternalAccessible := 'False'; ExternalVisible := 'False'; ExternalWritable := 'False'} : Real := 0.0;   // energy meter apparent power use rate1
      E_Apparent_Rate2_Import { ExternalAccessible := 'False'; ExternalVisible := 'False'; ExternalWritable := 'False'} : Real := 0.0;   // energy meter apparent power use rate2 Reset Time Energy
      R_Year_Energy { ExternalAccessible := 'False'; ExternalVisible := 'False'; ExternalWritable := 'False'} : Int := 0;   // Reset Energy year
      R_Month_Energy { ExternalAccessible := 'False'; ExternalVisible := 'False'; ExternalWritable := 'False'} : Int := 0;   // Reset Energy month
      R_Day_Energy { ExternalAccessible := 'False'; ExternalVisible := 'False'; ExternalWritable := 'False'} : Int := 0;   // Reset Energy day
      R_Hour_Energy { ExternalAccessible := 'False'; ExternalVisible := 'False'; ExternalWritable := 'False'} : Int := 0;   // Reset Energy hour
      R_Minute_Energy { ExternalAccessible := 'False'; ExternalVisible := 'False'; ExternalWritable := 'False'} : Int := 0;   // Reset Energy minute
      R_Second_Energy { ExternalAccessible := 'False'; ExternalVisible := 'False'; ExternalWritable := 'False'} : Int := 0;   // Reset Energy Second Rest Time Value
      R_Year_Value { ExternalAccessible := 'False'; ExternalVisible := 'False'; ExternalWritable := 'False'} : Int := 0;   // Reset Value year
      R_Month_Value { ExternalAccessible := 'False'; ExternalVisible := 'False'; ExternalWritable := 'False'} : Int := 0;   // Reset Value month
      R_Day_Value { ExternalAccessible := 'False'; ExternalVisible := 'False'; ExternalWritable := 'False'} : Int := 0;   // Reset Value day
      R_Hour_Value { ExternalAccessible := 'False'; ExternalVisible := 'False'; ExternalWritable := 'False'} : Int := 0;   // Reset Value hour
      R_Minute_Value { ExternalAccessible := 'False'; ExternalVisible := 'False'; ExternalWritable := 'False'} : Int := 0;   // Reset Value minute
      R_Second_Value { ExternalAccessible := 'False'; ExternalVisible := 'False'; ExternalWritable := 'False'} : Int := 0;   // Reset Value Second choice measuring unit
      Auto_Unit { ExternalAccessible := 'False'; ExternalVisible := 'False'; ExternalWritable := 'False'} : Bool := TRUE;
      C_U_Unit { ExternalAccessible := 'False'; ExternalVisible := 'False'; ExternalWritable := 'False'} : Int := 2;   // choiceVoltageUnit
      C_I_Unit { ExternalAccessible := 'False'; ExternalVisible := 'False'; ExternalWritable := 'False'} : Int := 2;   // choiceCurrentUnit
      C_S_Unit { ExternalAccessible := 'False'; ExternalVisible := 'False'; ExternalWritable := 'False'} : Int := 1;   // choiceApparentPowerUnit
      C_P_Unit { ExternalAccessible := 'False'; ExternalVisible := 'False'; ExternalWritable := 'False'} : Int := 1;   // choiceActivePowerUnit
      C_Q_Unit { ExternalAccessible := 'False'; ExternalVisible := 'False'; ExternalWritable := 'False'} : Int := 1;   // choiceReactivePowerUnit
      C_E_S_Unit { ExternalAccessible := 'False'; ExternalVisible := 'False'; ExternalWritable := 'False'} : Int := 1;   // choiceApparentEnergyUnit
      C_E_P_Unit { ExternalAccessible := 'False'; ExternalVisible := 'False'; ExternalWritable := 'False'} : Int := 1;   // choiceActiveEnergyUnit
      C_E_Q_Unit { ExternalAccessible := 'False'; ExternalVisible := 'False'; ExternalWritable := 'False'} : Int := 1;   // choiceReactiveEnergyUnit handing over value to visible at view
      V_Add_Value_Count { ExternalAccessible := 'False'; ExternalVisible := 'False'; ExternalWritable := 'False'} : Word := WORD#16#0000;   // counter add value
      U_PH_PH_Mod { ExternalAccessible := 'False'; ExternalVisible := 'False'; ExternalWritable := 'False'} : Word := WORD#16#0000;   // selection of voltage PH-PH show modification
      U_PH_N_Mod { ExternalAccessible := 'False'; ExternalVisible := 'False'; ExternalWritable := 'False'} : Word := WORD#16#0000;   // selection of voltage PH-N show modification
      I_Mod { ExternalAccessible := 'False'; ExternalVisible := 'False'; ExternalWritable := 'False'} : Word := WORD#16#0000;   // selection of current show modification
      S_Mod { ExternalAccessible := 'False'; ExternalVisible := 'False'; ExternalWritable := 'False'} : Word := WORD#16#0000;   // selection of apparent power show modification
      P_Mod { ExternalAccessible := 'False'; ExternalVisible := 'False'; ExternalWritable := 'False'} : Word := WORD#16#0000;   // selection of active power show modification
      Q_Mod { ExternalAccessible := 'False'; ExternalVisible := 'False'; ExternalWritable := 'False'} : Word := WORD#16#0000;   // selection of reactive power show modification
      E_Mod { ExternalAccessible := 'False'; ExternalVisible := 'False'; ExternalWritable := 'False'} : Word := WORD#16#0000;   // selection of energy meter show modification
      f_Mod { ExternalAccessible := 'False'; ExternalVisible := 'False'; ExternalWritable := 'False'} : Word := WORD#16#0000;   // selection of frequenz show modification
      Cos_Mod { ExternalAccessible := 'False'; ExternalVisible := 'False'; ExternalWritable := 'False'} : Word := WORD#16#0000;   // selection of efficiency factor show modification show value calculate
      Calculate_Value1 { ExternalAccessible := 'False'; ExternalVisible := 'False'; ExternalWritable := 'False'} : Word := WORD#16#0000;   // calculate value 1
      Calculate_Value2 { ExternalAccessible := 'False'; ExternalVisible := 'False'; ExternalWritable := 'False'} : Word := WORD#16#0000;   // calculate value 2
      Calculate_Value3 { ExternalAccessible := 'False'; ExternalVisible := 'False'; ExternalWritable := 'False'} : Word := WORD#16#0000;   // calculate value 3
      Calculate_Value4 { ExternalAccessible := 'False'; ExternalVisible := 'False'; ExternalWritable := 'False'} : Word := WORD#16#0000;   // calculate value 4
      Calculate_Value5 { ExternalAccessible := 'False'; ExternalVisible := 'False'; ExternalWritable := 'False'} : Word := WORD#16#0000;   // calculate value 5
      Calculate_Value6 { ExternalAccessible := 'False'; ExternalVisible := 'False'; ExternalWritable := 'False'} : Word := WORD#16#0000;   // calculate value 6 choice measuring unit
      U_Unit { ExternalAccessible := 'False'; ExternalVisible := 'False'; ExternalWritable := 'False'} : String[10];   // selection unit voltage
      I_Unit { ExternalAccessible := 'False'; ExternalVisible := 'False'; ExternalWritable := 'False'} : String[10];   // selection unit Current
      S_Unit { ExternalAccessible := 'False'; ExternalVisible := 'False'; ExternalWritable := 'False'} : String[10];   // selection unit ApparentPower
      P_Unit { ExternalAccessible := 'False'; ExternalVisible := 'False'; ExternalWritable := 'False'} : String[10];   // selection unit ActivePower
      Q_Unit { ExternalAccessible := 'False'; ExternalVisible := 'False'; ExternalWritable := 'False'} : String[10];   // selection unit ReactivePower
      S_Energy_Unit { ExternalAccessible := 'False'; ExternalVisible := 'False'; ExternalWritable := 'False'} : String[10];   // selection unit ApparentEnergy
      P_Energy_Unit { ExternalAccessible := 'False'; ExternalVisible := 'False'; ExternalWritable := 'False'} : String[10];   // selection unit ActiveEnergy
      Q_Energy_Unit { ExternalAccessible := 'False'; ExternalVisible := 'False'; ExternalWritable := 'False'} : String[10];   // selection unit ReactiveEnergy scale final value
      Scale_End_S { ExternalAccessible := 'False'; ExternalVisible := 'False'; ExternalWritable := 'False'} : Real := 0.0;   // scale final value ApparentPower
      Scale_End_P { ExternalAccessible := 'False'; ExternalVisible := 'False'; ExternalWritable := 'False'} : Real := 0.0;   // scale final value ActivePower
      Scale_End_Q { ExternalAccessible := 'False'; ExternalVisible := 'False'; ExternalWritable := 'False'} : Real := 0.0;   // scale final value ReactivePower max
      Scale_Begin_Q { ExternalAccessible := 'False'; ExternalVisible := 'False'; ExternalWritable := 'False'} : Real := 0.0;   // scale final value ReactivePower min
      Scale_End_I { ExternalAccessible := 'False'; ExternalVisible := 'False'; ExternalWritable := 'False'} : Real := 0.0;   // scale final value Current
      Scale_End_U_PH_PH { ExternalAccessible := 'False'; ExternalVisible := 'False'; ExternalWritable := 'False'} : Real := 0.0;   // scale final value voltage PH-PH
      Scale_End_U_PH_N { ExternalAccessible := 'False'; ExternalVisible := 'False'; ExternalWritable := 'False'} : Real := 0.0;   // scale final value voltage PH-N read value from AS
      Read_Value { ExternalAccessible := 'False'; ExternalVisible := 'False'; ExternalWritable := 'False'} : Bool := FALSE;   // HMI_Bits (STRUCT)
      HMI_Bits { ExternalAccessible := 'False'; ExternalVisible := 'False'; ExternalWritable := 'False'} : Struct   // return to driver
         Start_Acyclic { ExternalAccessible := 'False'; ExternalVisible := 'False'; ExternalWritable := 'False'} : Bool := FALSE;
         Start_Auto { ExternalAccessible := 'False'; ExternalVisible := 'False'; ExternalWritable := 'False'} : Bool := FALSE;
         Reset_min_max_Data { ExternalAccessible := 'False'; ExternalVisible := 'False'; ExternalWritable := 'False'} : Bool := FALSE;
         Reset_Energy_Meter { ExternalAccessible := 'False'; ExternalVisible := 'False'; ExternalWritable := 'False'} : Bool := FALSE;   // error code
      END_STRUCT;
      ERROR { ExternalAccessible := 'False'; ExternalVisible := 'False'; ExternalWritable := 'False'} : DWord := DWORD#16#0000_0000;   // error code
      Connection_Type { ExternalAccessible := 'False'; ExternalVisible := 'False'; ExternalWritable := 'False'} : Int;   // connection type of the measuring
      Driver_Error { ExternalAccessible := 'False'; ExternalVisible := 'False'; ExternalWritable := 'False'} : Int;   // error in driver detected================================================================================================================================static variable=================================================================================================================================================================================================================== temp value for calculation
   END_VAR
   VAR_IN_OUT
      Driver_Data : Struct   // Driver_Data (STRUCT)
         U_L1_L2 : Real;   // voltage L1-L2
         U_L2_L3 : Real;   // voltage L2-L3
         U_L3_L1 : Real;   // voltage L3-L1
         U_L1 : Real;   // voltage L1-N
         U_L2 : Real;   // voltage L2-N
         U_L3 : Real;   // voltage L3-N
         U_L1_L2_min : Real;   // minimum voltage U1 (PH-PH)
         U_L2_L3_min : Real;   // minimum voltage U2 (PH-PH)
         U_L3_L1_min : Real;   // minimum voltage U3 (PH-PH)
         U_L1_min : Real;   // minimum voltage U1 (PH-N)
         U_L2_min : Real;   // minimum voltage U2 (PH-N)
         U_L3_min : Real;   // minimum voltage U3 (PH-N)
         U_L1_L2_max : Real;   // maximum voltage U1 (PH-PH)
         U_L2_L3_max : Real;   // maximum voltage U2 (PH-PH)
         U_L3_L1_max : Real;   // maximum voltage U3 (PH-PH)
         U_L1_max : Real;   // maximum voltage U1 (PH-N)
         U_L2_max : Real;   // maximum voltage U2 (PH-N)
         U_L3_max : Real;   // maximum voltage U3 (PH-N)
         U_PH_PH_Average : Real;   // averagevoltage PH-PH
         U_PH_N_Average : Real;   // averagevoltage PH-N
         U_PH_PH_Average_min : Real;   // minimum averagevoltage PH-PH
         U_PH_N_Average_min : Real;   // minimum averagevoltage PH-N
         U_PH_PH_Average_max : Real;   // maximum averagevoltage PH-PH
         U_PH_N_Average_max : Real;   // maximum averagevoltage PH-N
         I_L1 : Real;   // current I1
         I_L2 : Real;   // current I2
         I_L3 : Real;   // current I3
         I_L1_min : Real;   // minimum current I1
         I_L2_min : Real;   // minimum current I2
         I_L3_min : Real;   // minimum current I3
         I_L1_max : Real;   // maximum current I1
         I_L2_max : Real;   // maximum current I2
         I_L3_max : Real;   // maximum current I3
         I_Average : Real;   // average currentI
         I_Average_min : Real;   // minimum average currentI
         I_Average_max : Real;   // maximum average currentI
         f : Real;   // frequency
         f_min : Real;   // minimum frequency
         f_max : Real;   // maximum frequency
         S_Total : Real;   // total apparent power
         S_Total_min : Real;   // minimum total apparent power
         S_Total_max : Real;   // maximum total apparent power
         P_Total : Real;   // total active power
         P_Total_min : Real;   // minimum total active power
         P_Total_max : Real;   // maximum total active power
         Q_Total : Real;   // total reactive power
         Q_Total_min : Real;   // minimum total power
         Q_Total_max : Real;   // maximum total power
         Cos_L1 : Real;   // power factor L1
         Cos_L1_min : Real;   // minimum power factor L1
         Cos_L1_max : Real;   // maximum power factor L1
         Cos_L2 : Real;   // power factor L2
         Cos_L2_min : Real;   // minimum power factor L2
         Cos_L2_max : Real;   // maximum power factor L2
         Cos_L3 : Real;   // power factor L3
         Cos_L3_min : Real;   // minimum power factor L3
         Cos_L3_max : Real;   // maximum power factor L3
         Cos_Total : Real;   // total power factor
         Cos_Total_min : Real;   // minimum total power factor
         Cos_Total_max : Real;   // maximum total power factor
         S_L1 : Real;   // apparent power S1
         S_L2 : Real;   // apparent power S2
         S_L3 : Real;   // apparent power S3
         S_L1_min : Real;   // minimum apparent power S1
         S_L2_min : Real;   // minimum apparent power S2
         S_L3_min : Real;   // minimum apparent power S3
         S_L1_max : Real;   // maximum apparent power S1
         S_L2_max : Real;   // maximum apparent power S2
         S_L3_max : Real;   // maximum apparent power S3
         P_L1 : Real;   // reactive active power P1
         P_L2 : Real;   // reactive active power P2
         P_L3 : Real;   // reactive active power P3
         P_L1_min : Real;   // minimum active power P1
         P_L2_min : Real;   // minimum active power P2
         P_L3_min : Real;   // minimum active power P3
         P_L1_max : Real;   // maximum active power P1
         P_L2_max : Real;   // maximum active power P2
         P_L3_max : Real;   // maximum active power P3
         Q_L1 : Real;   // reactive_power Q1
         Q_L2 : Real;   // reactive_power Q2
         Q_L3 : Real;   // reactive_power Q3
         Q_L1_min : Real;   // minimum reactive_power Q1
         Q_L2_min : Real;   // minimum reactive_power Q2
         Q_L3_min : Real;   // minimum reactive_power Q3
         Q_L1_max : Real;   // maximum reactive_power Q1
         Q_L2_max : Real;   // maximum reactive_power Q2
         Q_L3_max : Real;   // maximum reactive_power Q3
         E_Active_Rate1_Import : Real;   // energy meter active power use rate1
         E_Active_Rate2_Import : Real;   // energy meter active power use rate2
         E_Active_Rate1_Export : Real;   // energy meter active power export rate1
         E_Active_Rate2_Export : Real;   // energy meter active power export rate2
         E_Reactive_Rate1_Import : Real;   // energy meter reactive power use rate1
         E_Reactive_Rate2_Import : Real;   // energy meter reactive power use rate2
         E_Reactive_Rate1_Export : Real;   // energy meter reactive power export rate1
         E_Reactive_Rate2_Export : Real;   // energy meter reactive power export rate2
         E_Apparent_Rate1_Import : Real;   // energy meter apparent power use rate1
         E_Apparent_Rate2_Import : Real;   // energy meter apparent power use rate2
         RTime_Data_Energy : Date_And_Time;   // Resettime power
         RTime_Data_Value : Date_And_Time;   // Resettime value
         U_PH_PH_Mod : Word;   // voltage PH-PH show modification
         U_PH_N_Mod : Word;   // voltage PH-N show modification
         I_Mod : Word;   // current show modification
         S_Mod : Word;   // apparent power show modification
         P_Mod : Word;   // active power show modification
         Q_Mod : Word;   // reactive power show modification
         E_Mod : Word;   // energy meter show modification
         f_Mod : Word;   // frequenz show modification
         Cos_Mod : Word;   // efficiency factor show modification
         Calculate_Value1 : Word;   // calculate value 1
         Calculate_Value2 : Word;   // calculate value 2
         Calculate_Value3 : Word;   // calculate value 3
         Calculate_Value4 : Word;   // calculate value 4
         Calculate_Value5 : Word;   // calculate value 5
         Calculate_Value6 : Word;   // calculate value 6
         Energy_Meter_Unit : Word;   // energy meter unit
         Rest_Start_Auto : Bool;   // reset Auto start azyklisch
         Read_Value : Bool;   // read value (AS)
         Connection_Type : Int;   // connection type of the measuring
         Driver_Error : Int;   // error in driver detected================================================================================================================================output variablen================================================================================================================================================================================================================== energy value
      END_STRUCT;
   END_VAR
   VAR DB_SPECIFIC
      ZU_L1_L2 { ExternalAccessible := 'False'; ExternalVisible := 'False'; ExternalWritable := 'False'} : Real := 0.0;   // voltage L1-L2
      ZU_L2_L3 { ExternalAccessible := 'False'; ExternalVisible := 'False'; ExternalWritable := 'False'} : Real := 0.0;   // voltage L2-L3
      ZU_L3_L1 { ExternalAccessible := 'False'; ExternalVisible := 'False'; ExternalWritable := 'False'} : Real := 0.0;   // voltage L3-L1
      ZU_L1 { ExternalAccessible := 'False'; ExternalVisible := 'False'; ExternalWritable := 'False'} : Real := 0.0;   // voltage L1-N
      ZU_L2 { ExternalAccessible := 'False'; ExternalVisible := 'False'; ExternalWritable := 'False'} : Real := 0.0;   // voltage L2-N
      ZU_L3 { ExternalAccessible := 'False'; ExternalVisible := 'False'; ExternalWritable := 'False'} : Real := 0.0;   // voltage L3-N
      ZU_L1_L2_min { ExternalAccessible := 'False'; ExternalVisible := 'False'; ExternalWritable := 'False'} : Real := 0.0;   // minimum voltage U1 PH-PH
      ZU_L2_L3_min { ExternalAccessible := 'False'; ExternalVisible := 'False'; ExternalWritable := 'False'} : Real := 0.0;   // minimum voltage U2 PH-PH
      ZU_L3_L1_min { ExternalAccessible := 'False'; ExternalVisible := 'False'; ExternalWritable := 'False'} : Real := 0.0;   // minimum voltage U3 PH-PH
      ZU_L1_min { ExternalAccessible := 'False'; ExternalVisible := 'False'; ExternalWritable := 'False'} : Real := 0.0;   // minimum voltage U1 PH-N
      ZU_L2_min { ExternalAccessible := 'False'; ExternalVisible := 'False'; ExternalWritable := 'False'} : Real := 0.0;   // minimum voltage U2 PH-N
      ZU_L3_min { ExternalAccessible := 'False'; ExternalVisible := 'False'; ExternalWritable := 'False'} : Real := 0.0;   // minimum voltage U3 PH-N
      ZU_L1_L2_max { ExternalAccessible := 'False'; ExternalVisible := 'False'; ExternalWritable := 'False'} : Real := 0.0;   // maximum voltage U1 PH-PH
      ZU_L2_L3_max { ExternalAccessible := 'False'; ExternalVisible := 'False'; ExternalWritable := 'False'} : Real := 0.0;   // maximum voltage U2 PH-PH
      ZU_L3_L1_max { ExternalAccessible := 'False'; ExternalVisible := 'False'; ExternalWritable := 'False'} : Real := 0.0;   // maximum voltage U3 PH-PH
      ZU_L1_max { ExternalAccessible := 'False'; ExternalVisible := 'False'; ExternalWritable := 'False'} : Real := 0.0;   // maximum voltage U1 PH-N
      ZU_L2_max { ExternalAccessible := 'False'; ExternalVisible := 'False'; ExternalWritable := 'False'} : Real := 0.0;   // maximum voltage U2 PH-N
      ZU_L3_max { ExternalAccessible := 'False'; ExternalVisible := 'False'; ExternalWritable := 'False'} : Real := 0.0;   // maximum voltage U3 PH-N
      ZU_PH_PH_Average { ExternalAccessible := 'False'; ExternalVisible := 'False'; ExternalWritable := 'False'} : Real := 0.0;   // averagevoltage PH-PH
      ZU_PH_N_Average { ExternalAccessible := 'False'; ExternalVisible := 'False'; ExternalWritable := 'False'} : Real := 0.0;   // averagevoltage PH-N
      ZU_PH_PH_Average_min { ExternalAccessible := 'False'; ExternalVisible := 'False'; ExternalWritable := 'False'} : Real := 0.0;   // minimum averagevoltage PH-PH
      ZU_PH_N_Average_min { ExternalAccessible := 'False'; ExternalVisible := 'False'; ExternalWritable := 'False'} : Real := 0.0;   // minimum averagevoltage PH-N
      ZU_PH_PH_Average_max { ExternalAccessible := 'False'; ExternalVisible := 'False'; ExternalWritable := 'False'} : Real := 0.0;   // maximum averagevoltage PH-PH
      ZU_PH_N_Average_max { ExternalAccessible := 'False'; ExternalVisible := 'False'; ExternalWritable := 'False'} : Real := 0.0;   // maximum averagevoltage PH-N
      ZI_L1 { ExternalAccessible := 'False'; ExternalVisible := 'False'; ExternalWritable := 'False'} : Real := 0.0;   // current I1
      ZI_L2 { ExternalAccessible := 'False'; ExternalVisible := 'False'; ExternalWritable := 'False'} : Real := 0.0;   // current I2
      ZI_L3 { ExternalAccessible := 'False'; ExternalVisible := 'False'; ExternalWritable := 'False'} : Real := 0.0;   // current I3
      ZI_L1_min { ExternalAccessible := 'False'; ExternalVisible := 'False'; ExternalWritable := 'False'} : Real := 0.0;   // minimum current I1
      ZI_L2_min { ExternalAccessible := 'False'; ExternalVisible := 'False'; ExternalWritable := 'False'} : Real := 0.0;   // minimum current I2
      ZI_L3_min { ExternalAccessible := 'False'; ExternalVisible := 'False'; ExternalWritable := 'False'} : Real := 0.0;   // minimum current I3
      ZI_L1_max { ExternalAccessible := 'False'; ExternalVisible := 'False'; ExternalWritable := 'False'} : Real := 0.0;   // maximum current I1
      ZI_L2_max { ExternalAccessible := 'False'; ExternalVisible := 'False'; ExternalWritable := 'False'} : Real := 0.0;   // maximum current I2
      ZI_L3_max { ExternalAccessible := 'False'; ExternalVisible := 'False'; ExternalWritable := 'False'} : Real := 0.0;   // maximum current I3
      ZI_Average { ExternalAccessible := 'False'; ExternalVisible := 'False'; ExternalWritable := 'False'} : Real := 0.0;   // average currentI
      ZI_Average_min { ExternalAccessible := 'False'; ExternalVisible := 'False'; ExternalWritable := 'False'} : Real := 0.0;   // minimum average currentI
      ZI_Average_max { ExternalAccessible := 'False'; ExternalVisible := 'False'; ExternalWritable := 'False'} : Real := 0.0;   // maximum average currentI
      Zf { ExternalAccessible := 'False'; ExternalVisible := 'False'; ExternalWritable := 'False'} : Real := 0.0;   // frequency
      Zf_min { ExternalAccessible := 'False'; ExternalVisible := 'False'; ExternalWritable := 'False'} : Real := 0.0;   // minimum frequenz
      Zf_max { ExternalAccessible := 'False'; ExternalVisible := 'False'; ExternalWritable := 'False'} : Real := 0.0;   // maximum frequenz
      ZS_Total { ExternalAccessible := 'False'; ExternalVisible := 'False'; ExternalWritable := 'False'} : Real := 0.0;   // total apparent power
      ZS_Total_min { ExternalAccessible := 'False'; ExternalVisible := 'False'; ExternalWritable := 'False'} : Real := 0.0;   // minimum total apparent power
      ZS_Total_max { ExternalAccessible := 'False'; ExternalVisible := 'False'; ExternalWritable := 'False'} : Real := 0.0;   // maximum total apparent power
      ZP_Total { ExternalAccessible := 'False'; ExternalVisible := 'False'; ExternalWritable := 'False'} : Real := 0.0;   // total active power
      ZP_Total_min { ExternalAccessible := 'False'; ExternalVisible := 'False'; ExternalWritable := 'False'} : Real := 0.0;   // minimum total active power
      ZP_Total_max { ExternalAccessible := 'False'; ExternalVisible := 'False'; ExternalWritable := 'False'} : Real := 0.0;   // maximum total active power
      ZQ_Total { ExternalAccessible := 'False'; ExternalVisible := 'False'; ExternalWritable := 'False'} : Real := 0.0;   // total reactive power
      ZQ_Total_min { ExternalAccessible := 'False'; ExternalVisible := 'False'; ExternalWritable := 'False'} : Real := 0.0;   // minimum total reactive power
      ZQ_Total_max { ExternalAccessible := 'False'; ExternalVisible := 'False'; ExternalWritable := 'False'} : Real := 0.0;   // maximum total reactive power
      ZCos_Total { ExternalAccessible := 'False'; ExternalVisible := 'False'; ExternalWritable := 'False'} : Real := 0.0;   // total efficiency factor
      ZCos_Total_min { ExternalAccessible := 'False'; ExternalVisible := 'False'; ExternalWritable := 'False'} : Real := 0.0;   // minimum total power
      ZCos_Total_max { ExternalAccessible := 'False'; ExternalVisible := 'False'; ExternalWritable := 'False'} : Real := 0.0;   // maximum total power
      ZCos_L1 { ExternalAccessible := 'False'; ExternalVisible := 'False'; ExternalWritable := 'False'} : Real := 0.0;   // efficiency factor L1
      ZCos_L1_min { ExternalAccessible := 'False'; ExternalVisible := 'False'; ExternalWritable := 'False'} : Real := 0.0;   // minimum efficiency factor L1
      ZCos_L1_max { ExternalAccessible := 'False'; ExternalVisible := 'False'; ExternalWritable := 'False'} : Real := 0.0;   // maximum efficiency factor L1
      ZCos_L2 { ExternalAccessible := 'False'; ExternalVisible := 'False'; ExternalWritable := 'False'} : Real := 0.0;   // efficiency factor L2
      ZCos_L2_min { ExternalAccessible := 'False'; ExternalVisible := 'False'; ExternalWritable := 'False'} : Real := 0.0;   // minimum efficiency factor L2
      ZCos_L2_max { ExternalAccessible := 'False'; ExternalVisible := 'False'; ExternalWritable := 'False'} : Real := 0.0;   // maximum efficiency factor L2
      ZCOS_L3 { ExternalAccessible := 'False'; ExternalVisible := 'False'; ExternalWritable := 'False'} : Real := 0.0;   // efficiency factor L3
      ZCos_L3_min { ExternalAccessible := 'False'; ExternalVisible := 'False'; ExternalWritable := 'False'} : Real := 0.0;   // minimum efficiency factor L3
      ZCos_L3_max { ExternalAccessible := 'False'; ExternalVisible := 'False'; ExternalWritable := 'False'} : Real := 0.0;   // maximum efficiency factor L3
      ZS_L1 { ExternalAccessible := 'False'; ExternalVisible := 'False'; ExternalWritable := 'False'} : Real := 0.0;   // apparent power S1
      ZS_L2 { ExternalAccessible := 'False'; ExternalVisible := 'False'; ExternalWritable := 'False'} : Real := 0.0;   // apparent power S2
      ZS_L3 { ExternalAccessible := 'False'; ExternalVisible := 'False'; ExternalWritable := 'False'} : Real := 0.0;   // apparent power S3
      ZS_L1_min { ExternalAccessible := 'False'; ExternalVisible := 'False'; ExternalWritable := 'False'} : Real := 0.0;   // minimum apparent power S1
      ZS_L2_min { ExternalAccessible := 'False'; ExternalVisible := 'False'; ExternalWritable := 'False'} : Real := 0.0;   // minimum apparent power S2
      ZS_L3_min { ExternalAccessible := 'False'; ExternalVisible := 'False'; ExternalWritable := 'False'} : Real := 0.0;   // minimum apparent power S3
      ZS_L1_max { ExternalAccessible := 'False'; ExternalVisible := 'False'; ExternalWritable := 'False'} : Real := 0.0;   // maximum apparent power S1
      ZS_L2_max { ExternalAccessible := 'False'; ExternalVisible := 'False'; ExternalWritable := 'False'} : Real := 0.0;   // maximum apparent power S2
      ZS_L3_max { ExternalAccessible := 'False'; ExternalVisible := 'False'; ExternalWritable := 'False'} : Real := 0.0;   // maximum apparent power S3
      ZP_L1 { ExternalAccessible := 'False'; ExternalVisible := 'False'; ExternalWritable := 'False'} : Real := 0.0;   // reactive active power P1
      ZP_L2 { ExternalAccessible := 'False'; ExternalVisible := 'False'; ExternalWritable := 'False'} : Real := 0.0;   // reactive active power P2
      ZP_L3 { ExternalAccessible := 'False'; ExternalVisible := 'False'; ExternalWritable := 'False'} : Real := 0.0;   // reactive active power P3
      ZP_L1_min { ExternalAccessible := 'False'; ExternalVisible := 'False'; ExternalWritable := 'False'} : Real := 0.0;   // minimum active power P1
      ZP_L2_min { ExternalAccessible := 'False'; ExternalVisible := 'False'; ExternalWritable := 'False'} : Real := 0.0;   // minimum active power P2
      ZP_L3_min { ExternalAccessible := 'False'; ExternalVisible := 'False'; ExternalWritable := 'False'} : Real := 0.0;   // minimum active power P3
      ZP_L1_max { ExternalAccessible := 'False'; ExternalVisible := 'False'; ExternalWritable := 'False'} : Real := 0.0;   // maximum active power P1
      ZP_L2_max { ExternalAccessible := 'False'; ExternalVisible := 'False'; ExternalWritable := 'False'} : Real := 0.0;   // maximum active power P2
      ZP_L3_max { ExternalAccessible := 'False'; ExternalVisible := 'False'; ExternalWritable := 'False'} : Real := 0.0;   // maximum active power P3
      ZQ_L1 { ExternalAccessible := 'False'; ExternalVisible := 'False'; ExternalWritable := 'False'} : Real := 0.0;   // reactive_power Q1
      ZQ_L2 { ExternalAccessible := 'False'; ExternalVisible := 'False'; ExternalWritable := 'False'} : Real := 0.0;   // reactive_power Q2
      ZQ_L3 { ExternalAccessible := 'False'; ExternalVisible := 'False'; ExternalWritable := 'False'} : Real := 0.0;   // reactive_power Q3
      ZQ_L1_min { ExternalAccessible := 'False'; ExternalVisible := 'False'; ExternalWritable := 'False'} : Real := 0.0;   // minimum reactive_power Q1
      ZQ_L2_min { ExternalAccessible := 'False'; ExternalVisible := 'False'; ExternalWritable := 'False'} : Real := 0.0;   // minimum reactive_power Q2
      ZQ_L3_min { ExternalAccessible := 'False'; ExternalVisible := 'False'; ExternalWritable := 'False'} : Real := 0.0;   // minimum reactive_power Q3
      ZQ_L1_max { ExternalAccessible := 'False'; ExternalVisible := 'False'; ExternalWritable := 'False'} : Real := 0.0;   // maximum reactive_power Q1
      ZQ_L2_max { ExternalAccessible := 'False'; ExternalVisible := 'False'; ExternalWritable := 'False'} : Real := 0.0;   // maximum reactive_power Q2
      ZQ_L3_max { ExternalAccessible := 'False'; ExternalVisible := 'False'; ExternalWritable := 'False'} : Real := 0.0;   // maximum reactive_power Q3
      ZE_Active_Rate1_Import { ExternalAccessible := 'False'; ExternalVisible := 'False'; ExternalWritable := 'False'} : Real := 0.0;   // energy meter active power use rate1
      ZE_Active_Rate2_Import { ExternalAccessible := 'False'; ExternalVisible := 'False'; ExternalWritable := 'False'} : Real := 0.0;   // energy meter active power use rate2
      ZE_Active_Rate1_Export { ExternalAccessible := 'False'; ExternalVisible := 'False'; ExternalWritable := 'False'} : Real := 0.0;   // energy meter active power export rate1
      ZE_Active_Rate2_Export { ExternalAccessible := 'False'; ExternalVisible := 'False'; ExternalWritable := 'False'} : Real := 0.0;   // energy meter active power export rate2
      ZE_Reactive_Rate1_Import { ExternalAccessible := 'False'; ExternalVisible := 'False'; ExternalWritable := 'False'} : Real := 0.0;   // energy meter reactive power use rate1
      ZE_Reactive_Rate2_Import { ExternalAccessible := 'False'; ExternalVisible := 'False'; ExternalWritable := 'False'} : Real := 0.0;   // energy meter reactive power use rate2
      ZE_Reactive_Rate1_Export { ExternalAccessible := 'False'; ExternalVisible := 'False'; ExternalWritable := 'False'} : Real := 0.0;   // energy meter reactive power export rate1
      ZE_Reactive_Rate2_Export { ExternalAccessible := 'False'; ExternalVisible := 'False'; ExternalWritable := 'False'} : Real := 0.0;   // energy meter reactive power export rate2
      ZE_Apparent_Rate1_Import { ExternalAccessible := 'False'; ExternalVisible := 'False'; ExternalWritable := 'False'} : Real := 0.0;   // energy meter apparent power use rate1
      ZE_Apparent_Rate2_Import { ExternalAccessible := 'False'; ExternalVisible := 'False'; ExternalWritable := 'False'} : Real := 0.0;   // energy meter apparent power use rate2
      ZScale_End_S { ExternalAccessible := 'False'; ExternalVisible := 'False'; ExternalWritable := 'False'} : DInt := 4;
      ZScale_End_P { ExternalAccessible := 'False'; ExternalVisible := 'False'; ExternalWritable := 'False'} : DInt := 4;
      ZScale_End_Q { ExternalAccessible := 'False'; ExternalVisible := 'False'; ExternalWritable := 'False'} : DInt := 4;
      ZScale_End_I { ExternalAccessible := 'False'; ExternalVisible := 'False'; ExternalWritable := 'False'} : DInt := 4;
      ZScale_End_U_PH_PH { ExternalAccessible := 'False'; ExternalVisible := 'False'; ExternalWritable := 'False'} : DInt := 4;
      ZScale_End_U_PH_N { ExternalAccessible := 'False'; ExternalVisible := 'False'; ExternalWritable := 'False'} : DInt := 4;   // return time and data
      RTime_Data_Energy { ExternalAccessible := 'False'; ExternalVisible := 'False'; ExternalWritable := 'False'} : Date_And_Time := DT#1990-01-01-00:00:00;
   END_VAR
   VAR
      ZRTime_Data_Energy AT RTime_Data_Energy : Array[1..8] of Byte;   // AT RTime_Data_Energy : ARRAY [1..8] OF BYTE ;
   END_VAR
   VAR DB_SPECIFIC
      RTime_Data_Value { ExternalAccessible := 'False'; ExternalVisible := 'False'; ExternalWritable := 'False'} : Date_And_Time := DT#1990-01-01-00:00:00;
   END_VAR
   VAR
      ZRTime_Data_Value AT RTime_Data_Value : Array[1..8] of Byte;   // AT RTime_Data_Value : ARRAY [1..8] OF BYTE ; Driver_Data a connect
   END_VAR
   VAR DB_SPECIFIC
      Driver_Data_Connect { ExternalAccessible := 'False'; ExternalVisible := 'False'; ExternalWritable := 'False'} : Bool := FALSE;
      ZEnergy_Meter_Unit { ExternalAccessible := 'False'; ExternalVisible := 'False'; ExternalWritable := 'False'} : Word := WORD#16#0000;
   END_VAR
   VAR
      VEnergy_Meter_Unit AT ZEnergy_Meter_Unit : Array[1..16] of Bool;   // AT ZEnergy_Meter_Unit : ARRAY [1..16] OF BOOL ; temp value vor if
   END_VAR
   VAR DB_SPECIFIC
      U_PH_PH { ExternalAccessible := 'False'; ExternalVisible := 'False'; ExternalWritable := 'False'} : Real := 4.0;   // run-value voltage PH-PH
      U_PH_N { ExternalAccessible := 'False'; ExternalVisible := 'False'; ExternalWritable := 'False'} : Real := 4.0;   // run-value voltage PH-N
      I { ExternalAccessible := 'False'; ExternalVisible := 'False'; ExternalWritable := 'False'} : Real := 4.0;   // run-value current
      S { ExternalAccessible := 'False'; ExternalVisible := 'False'; ExternalWritable := 'False'} : Real := 4.0;   // run-value apparent power
      P { ExternalAccessible := 'False'; ExternalVisible := 'False'; ExternalWritable := 'False'} : Real := 4.0;   // run-value active power
      Q { ExternalAccessible := 'False'; ExternalVisible := 'False'; ExternalWritable := 'False'} : Real := 4.0;   // run-value reactive power max
      Q_min { ExternalAccessible := 'False'; ExternalVisible := 'False'; ExternalWritable := 'False'} : Real := 4.0;   // run-value reactive power min temp error
      Fehler { ExternalAccessible := 'False'; ExternalVisible := 'False'; ExternalWritable := 'False'} : DWord := DWORD#16#0000_0000;   // ================================================================================================================================temp variable=====================================================================================================================================================================================================================
   END_VAR
   VAR_TEMP
      In_Out_Pointer : Any;
      VIn_Out_Pointer AT In_Out_Pointer : Struct   // AT In_Out_Pointer : STRUCT
         ID : Byte;   // length over buffers
         Typ : Byte;   // data type of the variable
         ANZ : Int;   // amount of elements of this data type
         DBN : Int;   // DB number of the storage
         PTR : DWord;   // offset in this DB pointer source
      END_STRUCT;
   END_VAR
   VAR CONSTANT
      THOUSAND : Int := 1000;
      MILLION : Real := 1000000.0;
      ZSCALE_END_SPQ1 : Int := 4;
      ZSCALE_END_SPQ2 : Int := 5;
      ZSCALE_END_SPQ3 : Int := 10;
      ZSCALE_END_SPQ4 : Int := 100;
      ZSCALE_END_I1 : Int := 4;
      ZSCALE_END_I2 : Int := 5;
      ZSCALE_END_I3 : Int := 10;
      ZSCALE_END_I4 : Int := 100;
      AREA_TO_THOUSAND : Int := 1000;
      AREA_TO_HUNDRED : Int := 100;
      AREA_TO_TEN : Int := 10;
      AREA_TO_ZERO : Int := 0;
      MIN_VALUE : Int := 1;
      MAX_VALUE : Int := 750;
      MIN_ENERGY_VALUE : Int := 1;
      MAX_ENERGY_VALUE : Real := 999999.0;
      FACTOR : Real := 1.2;   // factor for calculation scalar end valueERROR_ADD_VALUE_COUNT := 1001 ;=================================================================================================================================input variable=================================================================================================================================================================================================================== User Messwerte
   END_VAR
BEGIN
   //
   //======================================================================================================================
   //==========main program================================================================================================
   //======================================================================================================================
   // check if a value is connected to IN_OUT Driver_Data 
   #In_Out_Pointer := #Driver_Data;
   // check db number is 0 and db offset is 0
   IF ((#VIn_Out_Pointer.DBN = 0) AND (#VIn_Out_Pointer.PTR = 0)) THEN
       // structure is not connected
       #Driver_Data_Connect := FALSE;
   ELSE
       // structure is connected
       #Driver_Data_Connect := TRUE;
   END_IF;
   //======================================================================================================================
   //==========structur value to temp value==================================================================================
   //====================================================================================================================== 
   #ZU_L1_L2 := (#Driver_Data.U_L1_L2);                  // voltage L1-L2
   #ZU_L2_L3 := (#Driver_Data.U_L2_L3);                  // voltage L2-L3
   #ZU_L3_L1 := (#Driver_Data.U_L3_L1);                  // voltage L3-L1
   #ZU_L1 := (#Driver_Data.U_L1);                     // voltage L1-N
   #ZU_L2 := (#Driver_Data.U_L2);                     // voltage L2-N
   #ZU_L3 := (#Driver_Data.U_L3);                     // voltage L3-N
   #ZU_L1_L2_min := (#Driver_Data.U_L1_L2_min);              // minimum voltage L1-L2
   #ZU_L2_L3_min := (#Driver_Data.U_L2_L3_min);              // minimum voltage L2-L3
   #ZU_L3_L1_min := (#Driver_Data.U_L3_L1_min);              // minimum voltage L3-L1
   #ZU_L1_min := (#Driver_Data.U_L1_min);                 // minimum voltage L1-N
   #ZU_L2_min := (#Driver_Data.U_L2_min);                 // minimum voltage L2-N
   #ZU_L3_min := (#Driver_Data.U_L3_min);                 // minimum voltage L3-N
   #ZU_L1_L2_max := (#Driver_Data.U_L1_L2_max);              // maximum voltage L1-L2
   #ZU_L2_L3_max := (#Driver_Data.U_L2_L3_max);              // maximum voltage L2-L3
   #ZU_L3_L1_max := (#Driver_Data.U_L3_L1_max);              // maximum voltage L3-L1
   #ZU_L1_max := (#Driver_Data.U_L1_max);                 // maximum voltage L1-N
   #ZU_L2_max := (#Driver_Data.U_L2_max);                 // maximum voltage L2-N
   #ZU_L3_max := (#Driver_Data.U_L3_max);                 // maximum voltage L3-N
   #ZU_PH_PH_Average := (#Driver_Data.U_PH_PH_Average);          // averagevoltage PH-PH
   #ZU_PH_N_Average := (#Driver_Data.U_PH_N_Average);           // averagevoltage PH-N
   #ZU_PH_PH_Average_min := (#Driver_Data.U_PH_PH_Average_min);      // minimum averagevoltage PH-PH
   #ZU_PH_N_Average_min := (#Driver_Data.U_PH_N_Average_min);       // minimum averagevoltage PH-N
   #ZU_PH_PH_Average_max := (#Driver_Data.U_PH_PH_Average_max);      // maximum averagevoltage PH-PH
   #ZU_PH_N_Average_max := (#Driver_Data.U_PH_N_Average_max);       // maximum averagevoltage PH-N            
   #ZI_L1 := (#Driver_Data.I_L1);                     // current I1   
   #ZI_L2 := (#Driver_Data.I_L2);                     // current I2
   #ZI_L3 := (#Driver_Data.I_L3);                     // current I3
   #ZI_L1_min := (#Driver_Data.I_L1_min);                 // minimum current I1
   #ZI_L2_min := (#Driver_Data.I_L2_min);                 // minimum current I2
   #ZI_L3_min := (#Driver_Data.I_L3_min);                 // minimum current I3
   #ZI_L1_max := (#Driver_Data.I_L1_max);                 // maximum current I1
   #ZI_L2_max := (#Driver_Data.I_L2_max);                 // maximum current I2
   #ZI_L3_max := (#Driver_Data.I_L3_max);                 // maximum current I3   
   #ZI_Average := (#Driver_Data.I_Average);                // average currentI
   #ZI_Average_min := (#Driver_Data.I_Average_min);            // minimum average currentI
   #ZI_Average_max := (#Driver_Data.I_Average_max);            // maximum average currentI    
   #Zf := (#Driver_Data.f);                        // frequency 
   #Zf_min := (#Driver_Data.f_min);                    // minimum frequenz
   #Zf_max := (#Driver_Data.f_max);                    // maximum frequenz    
   #ZS_Total := (#Driver_Data.S_Total);                  // total apparent power
   #ZS_Total_min := (#Driver_Data.S_Total_min);              // minimum total apparent power
   #ZS_Total_max := (#Driver_Data.S_Total_max);              // maximum total apparent power
   #ZP_Total := (#Driver_Data.P_Total);                  // total active power
   #ZP_Total_min := (#Driver_Data.P_Total_min);              // minimum total active power
   #ZP_Total_max := (#Driver_Data.P_Total_max);              // maximum total active power  
   #ZQ_Total := (#Driver_Data.Q_Total);                  // total reactive power
   #ZQ_Total_min := (#Driver_Data.Q_Total_min);              // minimum total reactive power
   #ZQ_Total_max := (#Driver_Data.Q_Total_max);              // maximum total reactive power
   #ZCos_Total := (#Driver_Data.Cos_Total);                // total efficiency factor
   #ZCos_Total_min := (#Driver_Data.Cos_Total_min);            // minimum total efficiency factor
   #ZCos_Total_max := (#Driver_Data.Cos_Total_max);            // maximum total efficiency factor
   #ZCos_L1 := (#Driver_Data.Cos_L1);                   // efficiency factor L1       
   #ZCos_L1_min := (#Driver_Data.Cos_L1_min);               // minimum efficiency factor L1
   #ZCos_L1_max := (#Driver_Data.Cos_L1_max);               // maximum efficiency factor L1
   #ZCos_L2 := (#Driver_Data.Cos_L2);                   // efficiency factor L2
   #ZCos_L2_min := (#Driver_Data.Cos_L2_min);               // minimum efficiency factor L2
   #ZCos_L2_max := (#Driver_Data.Cos_L2_max);               // maximum efficiency factor L2
   #ZCOS_L3 := (#Driver_Data.Cos_L3);                   // efficiency factor L3
   #ZCos_L3_min := (#Driver_Data.Cos_L3_min);               // minimum efficiency factor L3
   #ZCos_L3_max := (#Driver_Data.Cos_L3_max);               // maximum efficiency factor L3
   #ZS_L1 := (#Driver_Data.S_L1);                     // apparent power S1
   #ZS_L2 := (#Driver_Data.S_L2);                     // apparent power S2
   #ZS_L3 := (#Driver_Data.S_L3);                     // apparent power S3
   #ZS_L1_min := (#Driver_Data.S_L1_min);                 // minimum apparent power S1
   #ZS_L2_min := (#Driver_Data.S_L2_min);                 // minimum apparent power S2
   #ZS_L3_min := (#Driver_Data.S_L3_min);                 // minimum apparent power S3
   #ZS_L1_max := (#Driver_Data.S_L1_max);                 // maximum apparent power S1
   #ZS_L2_max := (#Driver_Data.S_L2_max);                 // maximum apparent power S2
   #ZS_L3_max := (#Driver_Data.S_L3_max);                 // maximum apparent power S3
   #ZP_L1 := (#Driver_Data.P_L1);                     // reactive active power P1
   #ZP_L2 := (#Driver_Data.P_L2);                     // reactive active power P2
   #ZP_L3 := (#Driver_Data.P_L3);                     // reactive active power P3
   #ZP_L1_min := (#Driver_Data.P_L1_min);                 // minimum active power P1
   #ZP_L2_min := (#Driver_Data.P_L2_min);                 // minimum active power P2
   #ZP_L3_min := (#Driver_Data.P_L3_min);                 // minimum active power P3
   #ZP_L1_max := (#Driver_Data.P_L1_max);                 // maximum active power P1
   #ZP_L2_max := (#Driver_Data.P_L2_max);                 // maximum active power P2
   #ZP_L3_max := (#Driver_Data.P_L3_max);                 // maximum active power P3
   #ZQ_L1 := (#Driver_Data.Q_L1);                     // reactive_power Q1
   #ZQ_L2 := (#Driver_Data.Q_L2);                     // reactive_power Q2
   #ZQ_L3 := (#Driver_Data.Q_L3);                     // reactive_power Q3
   #ZQ_L1_min := (#Driver_Data.Q_L1_min);                 // minimum reactive_power Q1
   #ZQ_L2_min := (#Driver_Data.Q_L2_min);                 // minimum reactive_power Q2
   #ZQ_L3_min := (#Driver_Data.Q_L3_min);                 // minimum reactive_power Q3
   #ZQ_L1_max := (#Driver_Data.Q_L1_max);                 // maximum reactive_power Q1
   #ZQ_L2_max := (#Driver_Data.Q_L2_max);                 // maximum reactive_power Q2
   #ZQ_L3_max := (#Driver_Data.Q_L3_max);                 // maximum reactive_power Q3
   #ZE_Active_Rate1_Import := (#Driver_Data.E_Active_Rate1_Import);    // energy meter active power use rate1        
   #ZE_Active_Rate2_Import := (#Driver_Data.E_Active_Rate2_Import);    // energy meter active power use rate2
   #ZE_Active_Rate1_Export := (#Driver_Data.E_Active_Rate1_Export);    // energy meter active power export rate1
   #ZE_Active_Rate2_Export := (#Driver_Data.E_Active_Rate2_Export);    // energy meter active power export rate2 
   #ZE_Reactive_Rate1_Import := (#Driver_Data.E_Reactive_Rate1_Import);  // energy meter reactive power use rate1
   #ZE_Reactive_Rate2_Import := (#Driver_Data.E_Reactive_Rate2_Import);  // energy meter reactive power use rate2
   #ZE_Reactive_Rate1_Export := (#Driver_Data.E_Reactive_Rate1_Export);  // energy meter reactive power export rate1
   #ZE_Reactive_Rate2_Export := (#Driver_Data.E_Reactive_Rate2_Export);  // energy meter reactive power export rate2
   #ZE_Apparent_Rate1_Import := (#Driver_Data.E_Apparent_Rate1_Import);  // energy meter apparent power use rate1
   #ZE_Apparent_Rate2_Import := (#Driver_Data.E_Apparent_Rate2_Import);  // energy meter apparent power use rate2
   #ZEnergy_Meter_Unit := (#Driver_Data.Energy_Meter_Unit);
   #Connection_Type := (#Driver_Data.Connection_Type);              // connection type of the measuring
   #Driver_Error := (#Driver_Data.Driver_Error);                // error in driver detected
   //======================================================================================================================
   //==========choice add value count======================================================================================
   //======================================================================================================================
   // choice user value and change
   CASE #Add_Value_Count OF
       0:
           #V_Add_Value_Count := 0;
       1:
           #V_Add_Value_Count := 1;
       2:
           #V_Add_Value_Count := 3;
       3:
           #V_Add_Value_Count := 7;
       4:
           #V_Add_Value_Count := 15;
       5:
           #V_Add_Value_Count := 31;
       6:
           #V_Add_Value_Count := 63;
       7:
           #V_Add_Value_Count := 127;
       8:
           #V_Add_Value_Count := 255;
       9:
           #V_Add_Value_Count := 511;
       10:
           #V_Add_Value_Count := 1023;
       11:
           #V_Add_Value_Count := 2047;
       12:
           #V_Add_Value_Count := 4095;
       ELSE:
           #V_Add_Value_Count := 4095;             // by all other counter show all Add_Value_counter     
   END_CASE;
   //======================================================================================================================
   //==========choice units================================================================================================
   //======================================================================================================================
   // choice auto or manual unit  
   IF (#Auto_Unit = TRUE) THEN
       // selection voltage unit
       IF ((#U_L1_L2 > #MAX_VALUE) OR (#U_L2_L3 > #MAX_VALUE) OR (#U_L3_L1 > #MAX_VALUE) OR
           (#U_L1 > #MAX_VALUE) OR (#U_L2 > #MAX_VALUE) OR (#U_L3 > #MAX_VALUE) OR
           (#U_L1_L2_max > #MAX_VALUE) OR (#U_L2_L3_max > #MAX_VALUE) OR (#U_L3_L1_max > #MAX_VALUE) OR
           (#U_L1_max > #MAX_VALUE) OR (#U_L2_max > #MAX_VALUE) OR (#U_L3_max > #MAX_VALUE))
           AND (#C_U_Unit < 3) THEN
           #C_U_Unit := #C_U_Unit + 1;
       ELSIF ((#U_L1_L2 < #MIN_VALUE) AND (#U_L2_L3 < #MIN_VALUE) AND (#U_L3_L1 < #MIN_VALUE) AND
           (#U_L1 < #MIN_VALUE) AND (#U_L2 < #MIN_VALUE) AND (#U_L3 < #MIN_VALUE) AND
           (#U_L1_L2_max < #MIN_VALUE) AND (#U_L2_L3_max < #MIN_VALUE) AND (#U_L3_L1_max < #MIN_VALUE) AND
           (#U_L1_max < #MIN_VALUE) AND (#U_L2_max < #MIN_VALUE) AND (#U_L3_max < #MIN_VALUE))
           AND (#C_U_Unit > 1) THEN
           #C_U_Unit := #C_U_Unit - 1;
       ELSE
           ;
       END_IF;
       // selection current unit
       IF ((#I_L1 > #MAX_VALUE) OR (#I_L2 > #MAX_VALUE) OR (#I_L3 > #MAX_VALUE) OR
           (#I_L1_max > #MAX_VALUE) OR (#I_L2_max > #MAX_VALUE) OR (#I_L3_max > #MAX_VALUE))
           AND (#C_I_Unit < 3) THEN
           #C_I_Unit := #C_I_Unit + 1;
       ELSIF ((#I_L1 < #MIN_VALUE) AND (#I_L2 < #MIN_VALUE) AND (#I_L3 < #MIN_VALUE) AND
           (#I_L1_max < #MIN_VALUE) AND (#I_L2_max < #MIN_VALUE) AND (#I_L3_max < #MIN_VALUE))
           AND (#C_I_Unit > 1) THEN
           #C_I_Unit := #C_I_Unit - 1;
       ELSE
           ;
       END_IF;
       // selection apparent power unit
       IF ((#S_L1_max > #MAX_VALUE) OR (#S_L2_max > #MAX_VALUE) OR (#S_L3_max > #MAX_VALUE) OR (#S_Total_max > #MAX_VALUE) OR
           (#S_L1 > #MAX_VALUE) OR (#S_L2 > #MAX_VALUE) OR (#S_L3 > #MAX_VALUE) OR (#S_Total > #MAX_VALUE))
           AND (#C_S_Unit < 4) THEN
           #C_S_Unit := #C_S_Unit + 1;
       ELSIF ((#S_L1 < #MIN_VALUE) AND (#S_L2 < #MIN_VALUE) AND (#S_L3 < #MIN_VALUE) AND (#S_Total < #MIN_VALUE) AND
           (#S_L1_max < #MIN_VALUE) AND (#S_L2_max < #MIN_VALUE) AND (#S_L3_max < #MIN_VALUE) AND (#S_Total_max < #MIN_VALUE))
           AND (#C_S_Unit > 1) THEN
           #C_S_Unit := #C_S_Unit - 1;
       ELSE
           ;
       END_IF;
       // selection active power unit
       IF ((#P_L1 > #MAX_VALUE) OR (#P_L2 > #MAX_VALUE) OR (#P_L3 > #MAX_VALUE) OR (#P_Total > #MAX_VALUE) OR
           (#P_L1_max > #MAX_VALUE) OR (#P_L2_max > #MAX_VALUE) OR (#P_L3_max > #MAX_VALUE) OR (#P_Total_max > #MAX_VALUE))
           AND (#C_P_Unit < 4) THEN
           #C_P_Unit := #C_P_Unit + 1;
       ELSIF ((#P_L1 < #MIN_VALUE) AND (#P_L2 < #MIN_VALUE) AND (#P_L3 < #MIN_VALUE) AND (#P_Total < #MIN_VALUE) AND
           (#P_L1_max < #MIN_VALUE) AND (#P_L2_max < #MIN_VALUE) AND (#P_L3_max < #MIN_VALUE) AND (#P_Total_max < #MIN_VALUE))
           AND (#C_P_Unit > 1) THEN
           #C_P_Unit := #C_P_Unit - 1;
       ELSE
           ;
       END_IF;
       // selection reactive power unit
       IF ((#Q_L1 > #MAX_VALUE) OR (#Q_L2 > #MAX_VALUE) OR (#Q_L3 > #MAX_VALUE) OR (#Q_Total > #MAX_VALUE) OR
           (#Q_L1_max > #MAX_VALUE) OR (#Q_L2_max > #MAX_VALUE) OR (#Q_L3_max > #MAX_VALUE) OR (#Q_Total_max > #MAX_VALUE)) OR
           ((#Q_L1 < - #MAX_VALUE) OR (#Q_L2 < - #MAX_VALUE) OR (#Q_L3 < - #MAX_VALUE) OR (#Q_Total < - #MAX_VALUE) OR
           (#Q_L1_max < - #MAX_VALUE) OR (#Q_L2_max < - #MAX_VALUE) OR (#Q_L3_max < - #MAX_VALUE) OR (#Q_Total_max < - #MAX_VALUE))
           AND (#C_Q_Unit < 4) THEN
           #C_Q_Unit := #C_Q_Unit + 1;
       ELSIF ((#Q_L1 < #MIN_VALUE) AND (#Q_L2 < #MIN_VALUE) AND (#Q_L3 < #MIN_VALUE) AND (#Q_Total < #MIN_VALUE) AND
           (#Q_L1_max < #MIN_VALUE) AND (#Q_L2_max < #MIN_VALUE) AND (#Q_L3_max < #MIN_VALUE) AND (#Q_Total_max < #MIN_VALUE)) AND
           ((#Q_L1 < - #MIN_VALUE) AND (#Q_L2 < - #MIN_VALUE) AND (#Q_L3 < - #MIN_VALUE) AND (#Q_Total < - #MIN_VALUE) AND
           (#Q_L1_max < - #MIN_VALUE) AND (#Q_L2_max < - #MIN_VALUE) AND (#Q_L3_max < - #MIN_VALUE) AND (#Q_Total_max < - #MIN_VALUE))
           AND (#C_Q_Unit > 1) THEN
           #C_Q_Unit := #C_Q_Unit - 1;
       ELSE
           ;
       END_IF;
       // selection active energy unit 
       IF ((#E_Active_Rate1_Import > #MAX_ENERGY_VALUE) OR (#E_Active_Rate2_Import > #MAX_ENERGY_VALUE) OR
           (#E_Active_Rate1_Export > #MAX_ENERGY_VALUE) OR (#E_Active_Rate2_Export > #MAX_ENERGY_VALUE))
           AND (#C_E_P_Unit < 4) THEN
           #C_E_P_Unit := #C_E_P_Unit + 1;
       ELSIF ((#E_Active_Rate1_Import < #MIN_ENERGY_VALUE) AND (#E_Active_Rate2_Import < #MIN_ENERGY_VALUE) AND
           (#E_Active_Rate1_Export < #MIN_ENERGY_VALUE) AND (#E_Active_Rate2_Export < #MIN_ENERGY_VALUE))
           AND (#C_E_P_Unit > 1) THEN
           #C_E_P_Unit := #C_E_P_Unit - 1;
       ELSE
           ;
       END_IF;
       // selection reactive energy unit
       IF ((#E_Reactive_Rate1_Import > #MAX_ENERGY_VALUE) OR (#E_Reactive_Rate2_Import > #MAX_ENERGY_VALUE) OR
           (#E_Reactive_Rate1_Export > #MAX_ENERGY_VALUE) OR (#E_Reactive_Rate2_Export > #MAX_ENERGY_VALUE))
           AND (#C_E_Q_Unit < 4) THEN
